
// ===== library: MasterCopy "S7-1500_LAnyAxis_Blocks (Drop in folder "Program blocks")" =====

// folder: LAnyAxis_Blocks

FUNCTION_BLOCK "LAnyAxis_MC_Power"   // FB30000, SCL
TITLE = LAnyAxis_MC_Power
{ S7_Optimized_Access := 'TRUE' }
AUTHOR : tech.team.motioncontrol@siemens.com
FAMILY : AnyAxis
VERSION : 1.0
// Support: tech.team.motioncontrol@siemens.com 
// See corresponding MC_ instruction in TIA Portal help (information system)
   VAR_INPUT
      Axis : DB_ANY;   // See corresponding parameter of MC_ instruction in TIA Portal help (information system)
      Enable : Bool;   // See corresponding parameter of MC_ instruction in TIA Portal help (information system)
      StartMode : DInt := 1;   // See corresponding parameter of MC_ instruction in TIA Portal help (information system)
      StopMode : Int;   // See corresponding parameter of MC_ instruction in TIA Portal help (information system)
   END_VAR
   VAR_OUTPUT
      Status : Bool;   // See corresponding parameter of MC_ instruction in TIA Portal help (information system)
      Busy : Bool;   // See corresponding parameter of MC_ instruction in TIA Portal help (information system)
      Error : Bool;   // See corresponding parameter of MC_ instruction in TIA Portal help (information system)
      ErrorID : Word;   // See corresponding parameter of MC_ instruction in TIA Portal help (information system)
   END_VAR
   VAR
      instMC : MC_POWER;   // Instance of MC_Instruction
      statAxis : DB_ANY;   // Internal variable of axis
      statAxisType : Int;   // Actual state / axis type
   END_VAR
   VAR CONSTANT
      ERROR_INVALID_TECHNOLOGY_OBJECT : Word := 16#8002;   // See corresponding parameter of MC_ instruction in TIA Portal help (information system)
      IDLE : Int := 0;   // State idle
      INVALID_AXIS : Int := -1;   // Axis type: Invalid
      EXTERNAL_ENCODER : Int := 1;   // Axis type: External encoder
      SPEED_AXIS : Int := 2;   // Axis type: Speed axis
      POSITIONING_AXIS : Int := 3;   // Axis type: Positioning axis
      SYNCHRONOUS_AXIS : Int := 4;   // Axis type: Synchronous axis
   END_VAR
BEGIN
   REGION HEADER
     //================================================================================
     // SIEMENS AG
     // (c)Copyright 2020 All Rights Reserved
     //--------------------------------------------------------------------------------
     // Library: LAnyAxis 
     // Tested with: S7-1515-2 PN
     // Engineering: TIA Portal V16
     // Restrictions: -
     // Requirements: S7-1500 FW 2.8.1
     // Functionality: Conversion DB_ANY --> TO_Axis
     // Support: tech.team.motioncontrol@siemens.com
     // Note: Parameter comments are only available in language 'English (United States)'
     //--------------------------------------------------------------------------------
     // Change log table:
     // Version  Date        Expert in charge  Changes applied
     // 01.00.00 10.03.2020  RS                First released version
     //================================================================================
   END_REGION

   REGION ENABLE
     IF (#statAxisType = #IDLE) AND #Enable THEN
       // Check axis type
       CASE TypeOfDB(#Axis) OF
         TO_POSITIONINGAXIS:
           #statAxisType := #POSITIONING_AXIS;
           #statAxis := #Axis;

         TO_SYNCHRONOUSAXIS:
           #statAxisType := #SYNCHRONOUS_AXIS;
           #statAxis := #Axis;

         TO_SPEEDAXIS:
           #statAxisType := #SPEED_AXIS;
           #statAxis := #Axis;

         TO_EXTERNALENCODER:
           #statAxisType := #EXTERNAL_ENCODER;
           #statAxis := #Axis;
         ELSE
           #statAxisType := #INVALID_AXIS;
           #statAxis := 0;
       END_CASE;

     ELSIF NOT #Enable AND (#statAxisType = #INVALID_AXIS) THEN
       #statAxisType := #IDLE;

       // Outputs
       #Status := FALSE;
       #Busy := FALSE;
       #Error := FALSE;
       #ErrorID := 16#0000;
     END_IF;
   END_REGION

   CASE #statAxisType OF
     #IDLE:
       ;

     #POSITIONING_AXIS,
     #SYNCHRONOUS_AXIS,
     #SPEED_AXIS,
     #EXTERNAL_ENCODER:
       REGION VALID_AXIS
         // Inputs
         #instMC.Enable := #Enable;
         #instMC.StartMode := #StartMode;
         #instMC.StopMode := #StopMode;

         // Call of MC instruction
         CASE #statAxisType OF
           #POSITIONING_AXIS:
             "LAnyAxis_UnpubPowerPosAxis"(axis := #statAxis,
                                          instMC := #instMC);
           #SYNCHRONOUS_AXIS:
             "LAnyAxis_UnpubPowerSyncAxis"(axis := #statAxis,
                                           instMC := #instMC);
           #SPEED_AXIS:
             "LAnyAxis_UnpubPowerSpeedAxis"(axis := #statAxis,
                                            instMC := #instMC);
           #EXTERNAL_ENCODER:
             "LAnyAxis_UnpubPowerExtEncoder"(axis := #statAxis,
                                             instMC := #instMC);
         END_CASE;

         // Outputs
         #Status := #instMC.Status;
         #Busy := #instMC.Busy;
         #Error := #instMC.Error;
         #ErrorID := #instMC.ErrorId;

         // Status of MC instruction
         IF NOT #instMC.Busy
           AND NOT #instMC.Error
           AND NOT #instMC.Status
         THEN
           // Not active
           #statAxisType := #IDLE;
         END_IF;
       END_REGION

     ELSE
       REGION INVALID_AXIS
         // Outputs
         #Status := FALSE;
         #Busy := FALSE;
         #Error := TRUE;
         #ErrorID := #ERROR_INVALID_TECHNOLOGY_OBJECT;
       END_REGION
   END_CASE;
END_FUNCTION_BLOCK

FUNCTION_BLOCK "LAnyAxis_MC_Reset"   // FB30001, SCL
TITLE = LAnyAxis_MC_Reset
{ S7_Optimized_Access := 'TRUE' }
AUTHOR : tech.team.motioncontrol@siemens.com
FAMILY : AnyAxis
VERSION : 1.0
// Support: tech.team.motioncontrol@siemens.com 
// See corresponding MC_ instruction in TIA Portal help (information system)
   VAR_INPUT
      Axis : DB_ANY;   // See corresponding parameter of MC_ instruction in TIA Portal help (information system)
      Execute : Bool;   // See corresponding parameter of MC_ instruction in TIA Portal help (information system)
      Restart : Bool;   // See corresponding parameter of MC_ instruction in TIA Portal help (information system)
   END_VAR
   VAR_OUTPUT
      Done : Bool;   // See corresponding parameter of MC_ instruction in TIA Portal help (information system)
      Busy : Bool;   // See corresponding parameter of MC_ instruction in TIA Portal help (information system)
      CommandAborted : Bool;   // See corresponding parameter of MC_ instruction in TIA Portal help (information system)
      Error : Bool;   // See corresponding parameter of MC_ instruction in TIA Portal help (information system)
      ErrorID : Word;   // See corresponding parameter of MC_ instruction in TIA Portal help (information system)
   END_VAR
   VAR
      instMC : MC_RESET;   // Instance of MC_Instruction
      statExecuteOld : Bool;   // Old value of execute
      statAxis : DB_ANY;   // Internal variable of axis
      statAxisType : Int;   // Actual state / axis type
   END_VAR
   VAR CONSTANT
      ERROR_INVALID_TECHNOLOGY_OBJECT : Word := 16#8002;   // See corresponding parameter of MC_ instruction in TIA Portal help (information system)
      IDLE : Int := 0;   // State idle
      INVALID_AXIS : Int := -1;   // Axis type: Invalid
      EXTERNAL_ENCODER : Int := 1;   // Axis type: External encoder
      SPEED_AXIS : Int := 2;   // Axis type: Speed axis
      POSITIONING_AXIS : Int := 3;   // Axis type: Positioning axis
      SYNCHRONOUS_AXIS : Int := 4;   // Axis type: Synchronous axis
      PROXY : Int := 5;   // Axis type: Leading axis proxy
   END_VAR
BEGIN
   REGION HEADER
     //================================================================================
     // SIEMENS AG
     // (c)Copyright 2020 All Rights Reserved
     //--------------------------------------------------------------------------------
     // Library: LAnyAxis 
     // Tested with: S7-1515-2 PN
     // Engineering: TIA Portal V16
     // Restrictions: -
     // Requirements: S7-1500 FW 2.8.1
     // Functionality: Conversion DB_ANY --> TO_Axis
     // Support: tech.team.motioncontrol@siemens.com
     // Note: Parameter comments are only available in language 'English (United States)'
     //--------------------------------------------------------------------------------
     // Change log table:
     // Version  Date        Expert in charge  Changes applied
     // 01.00.00 10.03.2020  RS                First released version
     //================================================================================
   END_REGION

   REGION EXECUTE
     IF #Execute AND NOT #statExecuteOld THEN
       // Copy parameter
       #instMC.Restart := #Restart;

       // Check axis type
       CASE TypeOfDB(#Axis) OF
         TO_POSITIONINGAXIS:
           #statAxisType := #POSITIONING_AXIS;
           #statAxis := #Axis;

         TO_SYNCHRONOUSAXIS:
           #statAxisType := #SYNCHRONOUS_AXIS;
           #statAxis := #Axis;

         TO_EXTERNALENCODER:
           #statAxisType := #EXTERNAL_ENCODER;
           #statAxis := #Axis;

         TO_SPEEDAXIS:
           #statAxisType := #SPEED_AXIS;
           #statAxis := #Axis;

         ELSE
           #statAxisType := #INVALID_AXIS;
           #statAxis := 0;
       END_CASE;

     ELSIF NOT #Execute AND (#statAxisType = #INVALID_AXIS) THEN
       #statAxisType := #IDLE;

       // Outputs
       #Done := FALSE;
       #Busy := FALSE;
       #CommandAborted := FALSE;
       #Error := FALSE;
       #ErrorID := 16#0000;
     END_IF;

     // Edge detection
     #statExecuteOld := #Execute;
   END_REGION

   CASE #statAxisType OF
     #IDLE:
       ;

     #POSITIONING_AXIS,
     #SYNCHRONOUS_AXIS,
     #SPEED_AXIS,
     #EXTERNAL_ENCODER,
     #PROXY:
       REGION VALID_AXIS
         // Inputs
         #instMC.Execute := #Execute;

         // Call of MC instruction
         CASE #statAxisType OF
           #POSITIONING_AXIS:
             "LAnyAxis_UnpubResetPosAxis"(axis := #statAxis,
                                          instMC := #instMC);
           #SYNCHRONOUS_AXIS:
             "LAnyAxis_UnpubResetSyncAxis"(axis := #statAxis,
                                           instMC := #instMC);
           #SPEED_AXIS:
             "LAnyAxis_UnpubResetSpeedAxis"(axis := #statAxis,
                                            instMC := #instMC);
           #EXTERNAL_ENCODER:
             "LAnyAxis_UnpubResetExtEncoder"(axis := #statAxis,
                                             instMC := #instMC);
         END_CASE;

         // Outputs
         #Done := #instMC.Done;
         #Busy := #instMC.Busy;
         #CommandAborted := #instMC.CommandAborted;
         #Error := #instMC.Error;
         #ErrorID := #instMC.ErrorId;

         // Status of MC instruction
         IF NOT #instMC.Done
           AND NOT #instMC.Busy
           AND NOT #instMC.CommandAborted
           AND NOT #instMC.Error
         THEN
           // Not active
           #statAxisType := #IDLE;
         END_IF;
       END_REGION

     ELSE
       REGION INVALID_AXIS
         // Outputs
         #Done := FALSE;
         #Busy := FALSE;
         #CommandAborted := FALSE;
         #Error := TRUE;
         #ErrorID := #ERROR_INVALID_TECHNOLOGY_OBJECT;
       END_REGION
   END_CASE;
END_FUNCTION_BLOCK

FUNCTION_BLOCK "LAnyAxis_MC_Home"   // FB30002, SCL
TITLE = LAnyAxis_MC_Home
{ S7_Optimized_Access := 'TRUE' }
AUTHOR : tech.team.motioncontrol@siemens.com
FAMILY : AnyAxis
VERSION : 1.0
// Support: tech.team.motioncontrol@siemens.com 
// See corresponding MC_ instruction in TIA Portal help (information system)
   VAR_INPUT
      Axis : DB_ANY;   // See corresponding parameter of MC_ instruction in TIA Portal help (information system)
      Execute : Bool;   // See corresponding parameter of MC_ instruction in TIA Portal help (information system)
      Position : LReal;   // See corresponding parameter of MC_ instruction in TIA Portal help (information system)
      Mode : Int;   // See corresponding parameter of MC_ instruction in TIA Portal help (information system)
   END_VAR
   VAR_OUTPUT
      ReferenceMarkPosition : LReal;   // See corresponding parameter of MC_ instruction in TIA Portal help (information system)
      Done : Bool;   // See corresponding parameter of MC_ instruction in TIA Portal help (information system)
      Busy : Bool;   // See corresponding parameter of MC_ instruction in TIA Portal help (information system)
      CommandAborted : Bool;   // See corresponding parameter of MC_ instruction in TIA Portal help (information system)
      Error : Bool;   // See corresponding parameter of MC_ instruction in TIA Portal help (information system)
      ErrorID : Word;   // See corresponding parameter of MC_ instruction in TIA Portal help (information system)
   END_VAR
   VAR
      instMC : MC_HOME;   // Instance of MC_Instruction
      statExecuteOld : Bool;   // Old value of execute
      statAxis : DB_ANY;   // Internal variable of axis
      statAxisType : Int;   // Actual state / axis type
   END_VAR
   VAR CONSTANT
      ERROR_INVALID_TECHNOLOGY_OBJECT : Word := 16#8002;   // See corresponding parameter of MC_ instruction in TIA Portal help (information system)
      IDLE : Int := 0;   // State idle
      INVALID_AXIS : Int := -1;   // Axis type: Invalid
      EXTERNAL_ENCODER : Int := 1;   // Axis type: External encoder
      POSITIONING_AXIS : Int := 3;   // Axis type: Positioning axis
      SYNCHRONOUS_AXIS : Int := 4;   // Axis type: Synchronous axis
   END_VAR
BEGIN
   REGION HEADER
     //================================================================================
     // SIEMENS AG
     // (c)Copyright 2020 All Rights Reserved
     //--------------------------------------------------------------------------------
     // Library: LAnyAxis 
     // Tested with: S7-1515-2 PN
     // Engineering: TIA Portal V16
     // Restrictions: -
     // Requirements: S7-1500 FW 2.8.1
     // Functionality: Conversion DB_ANY --> TO_Axis
     // Support: tech.team.motioncontrol@siemens.com
     // Note: Parameter comments are only available in language 'English (United States)'
     //--------------------------------------------------------------------------------
     // Change log table:
     // Version  Date        Expert in charge  Changes applied
     // 01.00.00 10.03.2020  RS                First released version
     //================================================================================
   END_REGION

   REGION EXECUTE
     IF #Execute AND NOT #statExecuteOld THEN
       // Copy parameter
       #instMC.Position := #Position;
       #instMC.Mode := #Mode;

       // Check axis type
       CASE TypeOfDB(#Axis) OF
         TO_POSITIONINGAXIS:
           #statAxisType := #POSITIONING_AXIS;
           #statAxis := #Axis;

         TO_SYNCHRONOUSAXIS:
           #statAxisType := #SYNCHRONOUS_AXIS;
           #statAxis := #Axis;

         TO_EXTERNALENCODER:
           #statAxisType := #EXTERNAL_ENCODER;
           #statAxis := #Axis;

         ELSE
           #statAxisType := #INVALID_AXIS;
           #statAxis := 0;
       END_CASE;

     ELSIF NOT #Execute AND (#statAxisType = #INVALID_AXIS) THEN
       #statAxisType := #IDLE;

       // Outputs
       #Done := FALSE;
       #Busy := FALSE;
       #CommandAborted := FALSE;
       #Error := FALSE;
       #ErrorID := 16#0000;
     END_IF;

     // Edge detection
     #statExecuteOld := #Execute;
   END_REGION

   CASE #statAxisType OF
     #IDLE:
       ;

     #POSITIONING_AXIS,
     #SYNCHRONOUS_AXIS,
     #EXTERNAL_ENCODER:
       REGION VALID_AXIS
         // Inputs
         #instMC.Execute := #Execute;

         // Call of MC instruction
         CASE #statAxisType OF
           #POSITIONING_AXIS:
             "LAnyAxis_UnpubHomePosAxis"(axis := #statAxis,
                                         instMC := #instMC);
           #SYNCHRONOUS_AXIS:
             "LAnyAxis_UnpubHomeSyncAxis"(axis := #statAxis,
                                          instMC := #instMC);
           #EXTERNAL_ENCODER:
             "LAnyAxis_UnpubHomeExtEncoder"(axis := #statAxis,
                                            instMC := #instMC);
         END_CASE;

         // Outputs
         #ReferenceMarkPosition := #instMC.ReferenceMarkPosition;
         #Done := #instMC.Done;
         #Busy := #instMC.Busy;
         #CommandAborted := #instMC.CommandAborted;
         #Error := #instMC.Error;
         #ErrorID := #instMC.ErrorId;

         // Status of MC instruction
         IF NOT #instMC.Done
           AND NOT #instMC.Busy
           AND NOT #instMC.CommandAborted
           AND NOT #instMC.Error
         THEN
           // Not active
           #statAxisType := #IDLE;
         END_IF;
       END_REGION

     ELSE
       REGION INVALID_AXIS
         // Outputs
         #Done := FALSE;
         #Busy := FALSE;
         #CommandAborted := FALSE;
         #Error := TRUE;
         #ErrorID := #ERROR_INVALID_TECHNOLOGY_OBJECT;
       END_REGION
   END_CASE;
END_FUNCTION_BLOCK

FUNCTION_BLOCK "LAnyAxis_MC_Halt"   // FB30003, SCL
TITLE = LAnyAxis_MC_Halt
{ S7_Optimized_Access := 'TRUE' }
AUTHOR : tech.team.motioncontrol@siemens.com
FAMILY : AnyAxis
VERSION : 1.0
// Support: tech.team.motioncontrol@siemens.com 
// See corresponding MC_ instruction in TIA Portal help (information system)
   VAR_INPUT
      Axis : DB_ANY;   // See corresponding parameter of MC_ instruction in TIA Portal help (information system)
      Execute : Bool;   // See corresponding parameter of MC_ instruction in TIA Portal help (information system)
      Deceleration : LReal := -1.0;   // See corresponding parameter of MC_ instruction in TIA Portal help (information system)
      Jerk : LReal := -1.0;   // See corresponding parameter of MC_ instruction in TIA Portal help (information system)
      AbortAcceleration : Bool;   // See corresponding parameter of MC_ instruction in TIA Portal help (information system)
   END_VAR
   VAR_OUTPUT
      Done : Bool;   // See corresponding parameter of MC_ instruction in TIA Portal help (information system)
      Busy : Bool;   // See corresponding parameter of MC_ instruction in TIA Portal help (information system)
      CommandAborted : Bool;   // See corresponding parameter of MC_ instruction in TIA Portal help (information system)
      Error : Bool;   // See corresponding parameter of MC_ instruction in TIA Portal help (information system)
      ErrorID : Word;   // See corresponding parameter of MC_ instruction in TIA Portal help (information system)
   END_VAR
   VAR
      instMC : MC_HALT;   // Instance of MC_Instruction
      statExecuteOld : Bool;   // Old value of execute
      statAxis : DB_ANY;   // Internal variable of axis
      statAxisType : Int;   // Actual state / axis type
   END_VAR
   VAR CONSTANT
      ERROR_INVALID_TECHNOLOGY_OBJECT : Word := 16#8002;   // See corresponding parameter of MC_ instruction in TIA Portal help (information system)
      IDLE : Int := 0;   // State idle
      INVALID_AXIS : Int := -1;   // Axis type: Invalid
      SPEED_AXIS : Int := 2;   // Axis type: Speed axis
      POSITIONING_AXIS : Int := 3;   // Axis type: Positioning axis
      SYNCHRONOUS_AXIS : Int := 4;   // Axis type: Synchronous axis
   END_VAR
BEGIN
   REGION HEADER
     //================================================================================
     // SIEMENS AG
     // (c)Copyright 2020 All Rights Reserved
     //--------------------------------------------------------------------------------
     // Library: LAnyAxis 
     // Tested with: S7-1515-2 PN
     // Engineering: TIA Portal V16
     // Restrictions: -
     // Requirements: S7-1500 FW 2.8.1
     // Functionality: Conversion DB_ANY --> TO_Axis
     // Support: tech.team.motioncontrol@siemens.com
     // Note: Parameter comments are only available in language 'English (United States)'
     //--------------------------------------------------------------------------------
     // Change log table:
     // Version  Date        Expert in charge  Changes applied
     // 01.00.00 10.03.2020  RS                First released version
     //================================================================================
   END_REGION

   REGION EXECUTE
     IF #Execute AND NOT #statExecuteOld THEN
       // Copy parameter
       #instMC.Deceleration := #Deceleration;
       #instMC.Jerk := #Jerk;
       #instMC.AbortAcceleration := #AbortAcceleration;

       // Check axis type
       CASE TypeOfDB(#Axis) OF
         TO_POSITIONINGAXIS:
           #statAxisType := #POSITIONING_AXIS;
           #statAxis := #Axis;

         TO_SYNCHRONOUSAXIS:
           #statAxisType := #SYNCHRONOUS_AXIS;
           #statAxis := #Axis;

         TO_SPEEDAXIS:
           #statAxisType := #SPEED_AXIS;
           #statAxis := #Axis;

         ELSE
           #statAxisType := #INVALID_AXIS;
           #statAxis := 0;
       END_CASE;

     ELSIF NOT #Execute AND (#statAxisType = #INVALID_AXIS) THEN
       #statAxisType := #IDLE;

       // Outputs
       #Done := FALSE;
       #Busy := FALSE;
       #CommandAborted := FALSE;
       #Error := FALSE;
       #ErrorID := 16#0000;
     END_IF;

     // Edge detection
     #statExecuteOld := #Execute;
   END_REGION

   CASE #statAxisType OF
     #IDLE:
       ;

     #POSITIONING_AXIS,
     #SYNCHRONOUS_AXIS,
     #SPEED_AXIS:
       REGION VALID_AXIS
         // Inputs
         #instMC.Execute := #Execute;

         // Call of MC instruction
         CASE #statAxisType OF
           #POSITIONING_AXIS:
             "LAnyAxis_UnpubHaltPosAxis"(axis := #statAxis,
                                         instMC := #instMC);
           #SYNCHRONOUS_AXIS:
             "LAnyAxis_UnpubHaltSyncAxis"(axis := #statAxis,
                                          instMC := #instMC);
           #SPEED_AXIS:
             #instMC(Axis := #statAxis);
         END_CASE;

         // Outputs
         #Done := #instMC.Done;
         #Busy := #instMC.Busy;
         #CommandAborted := #instMC.CommandAborted;
         #Error := #instMC.Error;
         #ErrorID := #instMC.ErrorId;

         // Status of MC instruction
         IF NOT #instMC.Done
           AND NOT #instMC.Busy
           AND NOT #instMC.CommandAborted
           AND NOT #instMC.Error
         THEN
           // Not active
           #statAxisType := #IDLE;
         END_IF;
       END_REGION

     ELSE
       REGION INVALID_AXIS
         // Outputs
         #Done := FALSE;
         #Busy := FALSE;
         #CommandAborted := FALSE;
         #Error := TRUE;
         #ErrorID := #ERROR_INVALID_TECHNOLOGY_OBJECT;
       END_REGION
   END_CASE;
END_FUNCTION_BLOCK

FUNCTION_BLOCK "LAnyAxis_MC_MoveAbsolute"   // FB30004, SCL
TITLE = LAnyAxis_MC_MoveAbsolute
{ S7_Optimized_Access := 'TRUE' }
AUTHOR : tech.team.motioncontrol@siemens.com
FAMILY : AnyAxis
VERSION : 1.0
// Support: tech.team.motioncontrol@siemens.com 
// See corresponding MC_ instruction in TIA Portal help (information system)
   VAR_INPUT
      Axis : DB_ANY;   // See corresponding parameter of MC_ instruction in TIA Portal help (information system)
      Execute : Bool;   // See corresponding parameter of MC_ instruction in TIA Portal help (information system)
      Position : LReal;   // See corresponding parameter of MC_ instruction in TIA Portal help (information system)
      Velocity : LReal := -1.0;   // See corresponding parameter of MC_ instruction in TIA Portal help (information system)
      Acceleration : LReal := -1.0;   // See corresponding parameter of MC_ instruction in TIA Portal help (information system)
      Deceleration : LReal := -1.0;   // See corresponding parameter of MC_ instruction in TIA Portal help (information system)
      Jerk : LReal := -1.0;   // See corresponding parameter of MC_ instruction in TIA Portal help (information system)
      Direction : Int := 1;   // See corresponding parameter of MC_ instruction in TIA Portal help (information system)
   END_VAR
   VAR_OUTPUT
      Done : Bool;   // See corresponding parameter of MC_ instruction in TIA Portal help (information system)
      Busy : Bool;   // See corresponding parameter of MC_ instruction in TIA Portal help (information system)
      CommandAborted : Bool;   // See corresponding parameter of MC_ instruction in TIA Portal help (information system)
      Error : Bool;   // See corresponding parameter of MC_ instruction in TIA Portal help (information system)
      ErrorID : Word;   // See corresponding parameter of MC_ instruction in TIA Portal help (information system)
   END_VAR
   VAR
      instMC : MC_MOVEABSOLUTE;   // Instance of MC_Instruction
      statExecuteOld : Bool;   // Old value of execute
      statAxis : DB_ANY;   // Internal variable of axis
      statAxisType : Int;   // Actual state / axis type
   END_VAR
   VAR CONSTANT
      ERROR_INVALID_TECHNOLOGY_OBJECT : Word := 16#8002;   // See corresponding parameter of MC_ instruction in TIA Portal help (information system)
      IDLE : Int := 0;   // State idle
      INVALID_AXIS : Int := -1;   // Axis type: Invalid
      EXTERNAL_ENCODER : Int := 1;   // Axis type: External encoder
      POSITIONING_AXIS : Int := 3;   // Axis type: Positioning axis
      SYNCHRONOUS_AXIS : Int := 4;   // Axis type: Synchronous axis
   END_VAR
BEGIN
   REGION HEADER
     //================================================================================
     // SIEMENS AG
     // (c)Copyright 2020 All Rights Reserved
     //--------------------------------------------------------------------------------
     // Library: LAnyAxis 
     // Tested with: S7-1515-2 PN
     // Engineering: TIA Portal V16
     // Restrictions: -
     // Requirements: S7-1500 FW 2.8.1
     // Functionality: Conversion DB_ANY --> TO_Axis
     // Support: tech.team.motioncontrol@siemens.com
     // Note: Parameter comments are only available in language 'English (United States)'
     //--------------------------------------------------------------------------------
     // Change log table:
     // Version  Date        Expert in charge  Changes applied
     // 01.00.00 10.03.2020  RS                First released version
     //================================================================================
   END_REGION

   REGION EXECUTE
     IF #Execute AND NOT #statExecuteOld THEN
       // Copy parameter
       #instMC.Position := #Position;
       #instMC.Velocity := #Velocity;
       #instMC.Acceleration := #Acceleration;
       #instMC.Deceleration := #Deceleration;
       #instMC.Jerk := #Jerk;
       #instMC.Direction := #Direction;

       // Check axis type
       CASE TypeOfDB(#Axis) OF
         TO_POSITIONINGAXIS:
           #statAxisType := #POSITIONING_AXIS;
           #statAxis := #Axis;

         TO_SYNCHRONOUSAXIS:
           #statAxisType := #SYNCHRONOUS_AXIS;
           #statAxis := #Axis;

         ELSE
           #statAxisType := #INVALID_AXIS;
           #statAxis := 0;
       END_CASE;

     ELSIF NOT #Execute AND (#statAxisType = #INVALID_AXIS) THEN
       #statAxisType := #IDLE;

       // Outputs
       #Done := FALSE;
       #Busy := FALSE;
       #CommandAborted := FALSE;
       #Error := FALSE;
       #ErrorID := 16#0000;
     END_IF;

     // Edge detection
     #statExecuteOld := #Execute;
   END_REGION

   CASE #statAxisType OF
     #IDLE:
       ;

     #POSITIONING_AXIS,
     #SYNCHRONOUS_AXIS:
       REGION VALID_AXIS
         // Inputs
         #instMC.Execute := #Execute;

         // Call of MC instruction
         CASE #statAxisType OF
           #POSITIONING_AXIS:
             #instMC(Axis := #statAxis);
           #SYNCHRONOUS_AXIS:
             "LAnyAxis_UnpubMoveAbsoluteSyncAxis"(axis := #statAxis,
                                                  instMC := #instMC);
         END_CASE;

         // Outputs
         #Done := #instMC.Done;
         #Busy := #instMC.Busy;
         #CommandAborted := #instMC.CommandAborted;
         #Error := #instMC.Error;
         #ErrorID := #instMC.ErrorId;

         // Status of MC instruction
         IF NOT #instMC.Done
           AND NOT #instMC.Busy
           AND NOT #instMC.CommandAborted
           AND NOT #instMC.Error
         THEN
           // Not active
           #statAxisType := #IDLE;
         END_IF;
       END_REGION

     ELSE
       REGION INVALID_AXIS
         // Outputs
         #Done := FALSE;
         #Busy := FALSE;
         #CommandAborted := FALSE;
         #Error := TRUE;
         #ErrorID := #ERROR_INVALID_TECHNOLOGY_OBJECT;
       END_REGION
   END_CASE;
END_FUNCTION_BLOCK

FUNCTION_BLOCK "LAnyAxis_MC_MoveRelative"   // FB30005, SCL
TITLE = LAnyAxis_MC_MoveRelative
{ S7_Optimized_Access := 'TRUE' }
AUTHOR : tech.team.motioncontrol@siemens.com
FAMILY : AnyAxis
VERSION : 1.0
// Support: tech.team.motioncontrol@siemens.com 
// See corresponding MC_ instruction in TIA Portal help (information system)
   VAR_INPUT
      Axis : DB_ANY;   // See corresponding parameter of MC_ instruction in TIA Portal help (information system)
      Execute : Bool;   // See corresponding parameter of MC_ instruction in TIA Portal help (information system)
      Distance : LReal;   // See corresponding parameter of MC_ instruction in TIA Portal help (information system)
      Velocity : LReal := -1.0;   // See corresponding parameter of MC_ instruction in TIA Portal help (information system)
      Acceleration : LReal := -1.0;   // See corresponding parameter of MC_ instruction in TIA Portal help (information system)
      Deceleration : LReal := -1.0;   // See corresponding parameter of MC_ instruction in TIA Portal help (information system)
      Jerk : LReal := -1.0;   // See corresponding parameter of MC_ instruction in TIA Portal help (information system)
   END_VAR
   VAR_OUTPUT
      Done : Bool;   // See corresponding parameter of MC_ instruction in TIA Portal help (information system)
      Busy : Bool;   // See corresponding parameter of MC_ instruction in TIA Portal help (information system)
      CommandAborted : Bool;   // See corresponding parameter of MC_ instruction in TIA Portal help (information system)
      Error : Bool;   // See corresponding parameter of MC_ instruction in TIA Portal help (information system)
      ErrorID : Word;   // See corresponding parameter of MC_ instruction in TIA Portal help (information system)
   END_VAR
   VAR
      instMC : MC_MOVERELATIVE;   // Instance of MC_Instruction
      statExecuteOld : Bool;   // Old value of execute
      statAxis : DB_ANY;   // Internal variable of axis
      statAxisType : Int;   // Actual state / axis type
   END_VAR
   VAR CONSTANT
      ERROR_INVALID_TECHNOLOGY_OBJECT : Word := 16#8002;   // See corresponding parameter of MC_ instruction in TIA Portal help (information system)
      IDLE : Int := 0;   // State idle
      INVALID_AXIS : Int := -1;   // Axis type: Invalid
      POSITIONING_AXIS : Int := 3;   // Axis type: Positioning axis
      SYNCHRONOUS_AXIS : Int := 4;   // Axis type: Synchronous axis
   END_VAR
BEGIN
   REGION HEADER
     //================================================================================
     // SIEMENS AG
     // (c)Copyright 2020 All Rights Reserved
     //--------------------------------------------------------------------------------
     // Library: LAnyAxis 
     // Tested with: S7-1515-2 PN
     // Engineering: TIA Portal V16
     // Restrictions: -
     // Requirements: S7-1500 FW 2.8.1
     // Functionality: Conversion DB_ANY --> TO_Axis
     // Support: tech.team.motioncontrol@siemens.com
     // Note: Parameter comments are only available in language 'English (United States)'
     //--------------------------------------------------------------------------------
     // Change log table:
     // Version  Date        Expert in charge  Changes applied
     // 01.00.00 10.03.2020  RS                First released version
     //================================================================================
   END_REGION

   REGION EXECUTE
     IF #Execute AND NOT #statExecuteOld THEN
       // Copy parameter
       #instMC.Distance := #Distance;
       #instMC.Velocity := #Velocity;
       #instMC.Acceleration := #Acceleration;
       #instMC.Deceleration := #Deceleration;
       #instMC.Jerk := #Jerk;

       // Check axis type
       CASE TypeOfDB(#Axis) OF
         TO_POSITIONINGAXIS:
           #statAxisType := #POSITIONING_AXIS;
           #statAxis := #Axis;

         TO_SYNCHRONOUSAXIS:
           #statAxisType := #SYNCHRONOUS_AXIS;
           #statAxis := #Axis;

         ELSE
           #statAxisType := #INVALID_AXIS;
           #statAxis := 0;
       END_CASE;

     ELSIF NOT #Execute AND (#statAxisType = #INVALID_AXIS) THEN
       #statAxisType := #IDLE;

       // Outputs
       #Done := FALSE;
       #Busy := FALSE;
       #CommandAborted := FALSE;
       #Error := FALSE;
       #ErrorID := 16#0000;
     END_IF;

     // Edge detection
     #statExecuteOld := #Execute;
   END_REGION

   CASE #statAxisType OF
     #IDLE:
       ;

     #POSITIONING_AXIS,
     #SYNCHRONOUS_AXIS:
       REGION VALID_AXIS
         // Inputs
         #instMC.Execute := #Execute;

         // Call of MC instruction
         CASE #statAxisType OF
           #POSITIONING_AXIS:
             #instMC(Axis := #statAxis);
           #SYNCHRONOUS_AXIS:
             "LAnyAxis_UnpubMoveRelativeSyncAxis"(axis := #statAxis,
                                                  instMC := #instMC);
         END_CASE;

         // Outputs
         #Done := #instMC.Done;
         #Busy := #instMC.Busy;
         #CommandAborted := #instMC.CommandAborted;
         #Error := #instMC.Error;
         #ErrorID := #instMC.ErrorId;

         // Status of MC instruction
         IF NOT #instMC.Done
           AND NOT #instMC.Busy
           AND NOT #instMC.CommandAborted
           AND NOT #instMC.Error
         THEN
           // Not active
           #statAxisType := #IDLE;
         END_IF;
       END_REGION

     ELSE
       REGION INVALID_AXIS
         // Outputs
         #Done := FALSE;
         #Busy := FALSE;
         #CommandAborted := FALSE;
         #Error := TRUE;
         #ErrorID := #ERROR_INVALID_TECHNOLOGY_OBJECT;
       END_REGION
   END_CASE;
END_FUNCTION_BLOCK

FUNCTION_BLOCK "LAnyAxis_MC_MoveVelocity"   // FB30006, SCL
TITLE = LAnyAxis_MC_MoveVelocity
{ S7_Optimized_Access := 'TRUE' }
AUTHOR : tech.team.motioncontrol@siemens.com
FAMILY : AnyAxis
VERSION : 1.0
// Support: tech.team.motioncontrol@siemens.com 
// See corresponding MC_ instruction in TIA Portal help (information system)
   VAR_INPUT
      Axis : DB_ANY;   // See corresponding parameter of MC_ instruction in TIA Portal help (information system)
      Execute : Bool;   // See corresponding parameter of MC_ instruction in TIA Portal help (information system)
      Velocity : LReal := 100.0;   // See corresponding parameter of MC_ instruction in TIA Portal help (information system)
      Acceleration : LReal := -1.0;   // See corresponding parameter of MC_ instruction in TIA Portal help (information system)
      Deceleration : LReal := -1.0;   // See corresponding parameter of MC_ instruction in TIA Portal help (information system)
      Jerk : LReal := -1.0;   // See corresponding parameter of MC_ instruction in TIA Portal help (information system)
      Direction : Int;   // See corresponding parameter of MC_ instruction in TIA Portal help (information system)
      Current : Bool;   // See corresponding parameter of MC_ instruction in TIA Portal help (information system)
      PositionControlled : Bool := TRUE;   // See corresponding parameter of MC_ instruction in TIA Portal help (information system)
   END_VAR
   VAR_OUTPUT
      InVelocity : Bool;   // See corresponding parameter of MC_ instruction in TIA Portal help (information system)
      Busy : Bool;   // See corresponding parameter of MC_ instruction in TIA Portal help (information system)
      CommandAborted : Bool;   // See corresponding parameter of MC_ instruction in TIA Portal help (information system)
      Error : Bool;   // See corresponding parameter of MC_ instruction in TIA Portal help (information system)
      ErrorID : Word;   // See corresponding parameter of MC_ instruction in TIA Portal help (information system)
   END_VAR
   VAR
      instMC : MC_MOVEVELOCITY;   // Instance of MC_Instruction
      statExecuteOld : Bool;   // Old value of execute
      statAxis : DB_ANY;   // Internal variable of axis
      statAxisType : Int;   // Actual state / axis type
   END_VAR
   VAR CONSTANT
      ERROR_INVALID_TECHNOLOGY_OBJECT : Word := 16#8002;   // See corresponding parameter of MC_ instruction in TIA Portal help (information system)
      IDLE : Int := 0;   // State idle
      INVALID_AXIS : Int := -1;   // Axis type: Invalid
      SPEED_AXIS : Int := 2;   // Axis type: Speed axis
      POSITIONING_AXIS : Int := 3;   // Axis type: Positioning axis
      SYNCHRONOUS_AXIS : Int := 4;   // Axis type: Synchronous axis
   END_VAR
BEGIN
   REGION HEADER
     //================================================================================
     // SIEMENS AG
     // (c)Copyright 2020 All Rights Reserved
     //--------------------------------------------------------------------------------
     // Library: LAnyAxis 
     // Tested with: S7-1515-2 PN
     // Engineering: TIA Portal V16
     // Restrictions: -
     // Requirements: S7-1500 FW 2.8.1
     // Functionality: Conversion DB_ANY --> TO_Axis
     // Support: tech.team.motioncontrol@siemens.com
     // Note: Parameter comments are only available in language 'English (United States)'
     //--------------------------------------------------------------------------------
     // Change log table:
     // Version  Date        Expert in charge  Changes applied
     // 01.00.00 10.03.2020  RS                First released version
     //================================================================================
   END_REGION

   REGION EXECUTE
     IF #Execute AND NOT #statExecuteOld THEN
       // Copy parameter
       #instMC.Velocity := #Velocity;
       #instMC.Acceleration := #Acceleration;
       #instMC.Deceleration := #Deceleration;
       #instMC.Jerk := #Jerk;
       #instMC.Direction := #Direction;
       #instMC.Current := #Current;
       #instMC.PositionControlled := #PositionControlled;

       // Check axis type
       CASE TypeOfDB(#Axis) OF
         TO_POSITIONINGAXIS:
           #statAxisType := #POSITIONING_AXIS;
           #statAxis := #Axis;

         TO_SYNCHRONOUSAXIS:
           #statAxisType := #SYNCHRONOUS_AXIS;
           #statAxis := #Axis;

         TO_SPEEDAXIS:
           #statAxisType := #SPEED_AXIS;
           #statAxis := #Axis;

         ELSE
           #statAxisType := #INVALID_AXIS;
           #statAxis := 0;
       END_CASE;

     ELSIF NOT #Execute AND (#statAxisType = #INVALID_AXIS) THEN
       #statAxisType := #IDLE;

       // Outputs
       #InVelocity := FALSE;
       #Busy := FALSE;
       #CommandAborted := FALSE;
       #Error := FALSE;
       #ErrorID := 16#0000;
     END_IF;

     // Edge detection
     #statExecuteOld := #Execute;
   END_REGION

   CASE #statAxisType OF
     #IDLE:
       ;

     #POSITIONING_AXIS,
     #SYNCHRONOUS_AXIS,
     #SPEED_AXIS:
       REGION VALID_AXIS
         // Inputs
         #instMC.Execute := #Execute;

         // Call of MC instruction
         CASE #statAxisType OF
           #POSITIONING_AXIS:
             "LAnyAxis_UnpubMoveVelocityPosAxis"(axis := #statAxis,
                                                 instMC := #instMC);
           #SYNCHRONOUS_AXIS:
             "LAnyAxis_UnpubMoveVelocitySyncAxis"(axis := #statAxis,
                                                  instMC := #instMC);
           #SPEED_AXIS:
             #instMC(Axis := #statAxis);
         END_CASE;

         // Outputs
         #InVelocity := #instMC.InVelocity;
         #Busy := #instMC.Busy;
         #CommandAborted := #instMC.CommandAborted;
         #Error := #instMC.Error;
         #ErrorID := #instMC.ErrorId;

         // Status of MC instruction
         IF NOT #instMC.Busy
           AND NOT #instMC.CommandAborted
           AND NOT #instMC.Error
         THEN
           // Not active
           #statAxisType := #IDLE;
         END_IF;
       END_REGION

     ELSE
       REGION INVALID_AXIS
         // Outputs
         #InVelocity := FALSE;
         #Busy := FALSE;
         #CommandAborted := FALSE;
         #Error := TRUE;
         #ErrorID := #ERROR_INVALID_TECHNOLOGY_OBJECT;
       END_REGION
   END_CASE;
END_FUNCTION_BLOCK

FUNCTION_BLOCK "LAnyAxis_MC_MoveJog"   // FB30007, SCL
TITLE = LAnyAxis_MC_MoveJog
{ S7_Optimized_Access := 'TRUE' }
AUTHOR : tech.team.motioncontrol@siemens.com
FAMILY : AnyAxis
VERSION : 1.0
// Support: tech.team.motioncontrol@siemens.com 
// See corresponding MC_ instruction in TIA Portal help (information system)
   VAR_INPUT
      Axis : DB_ANY;   // See corresponding parameter of MC_ instruction in TIA Portal help (information system)
      JogForward : Bool;   // See corresponding parameter of MC_ instruction in TIA Portal help (information system)
      JogBackward : Bool;   // See corresponding parameter of MC_ instruction in TIA Portal help (information system)
      Velocity : LReal := 100.0;   // See corresponding parameter of MC_ instruction in TIA Portal help (information system)
      Acceleration : LReal := -1.0;   // See corresponding parameter of MC_ instruction in TIA Portal help (information system)
      Deceleration : LReal := -1.0;   // See corresponding parameter of MC_ instruction in TIA Portal help (information system)
      Jerk : LReal := -1.0;   // See corresponding parameter of MC_ instruction in TIA Portal help (information system)
      PositionControlled : Bool := TRUE;   // See corresponding parameter of MC_ instruction in TIA Portal help (information system)
   END_VAR
   VAR_OUTPUT
      InVelocity : Bool;   // See corresponding parameter of MC_ instruction in TIA Portal help (information system)
      Busy : Bool;   // See corresponding parameter of MC_ instruction in TIA Portal help (information system)
      CommandAborted : Bool;   // See corresponding parameter of MC_ instruction in TIA Portal help (information system)
      Error : Bool;   // See corresponding parameter of MC_ instruction in TIA Portal help (information system)
      ErrorID : Word;   // See corresponding parameter of MC_ instruction in TIA Portal help (information system)
   END_VAR
   VAR
      instMC : MC_MOVEJOG;   // Instance of MC_Instruction
      statAxis : DB_ANY;   // Internal variable of axis
      statAxisType : Int;   // Actual state / axis type
   END_VAR
   VAR CONSTANT
      ERROR_INVALID_TECHNOLOGY_OBJECT : Word := 16#8002;   // See corresponding parameter of MC_ instruction in TIA Portal help (information system)
      IDLE : Int := 0;   // State idle
      INVALID_AXIS : Int := -1;   // Axis type: Invalid
      SPEED_AXIS : Int := 2;   // Axis type: Speed axis
      POSITIONING_AXIS : Int := 3;   // Axis type: Positioning axis
      SYNCHRONOUS_AXIS : Int := 4;   // Axis type: Synchronous axis
   END_VAR
BEGIN
   REGION HEADER
     //================================================================================
     // SIEMENS AG
     // (c)Copyright 2020 All Rights Reserved
     //--------------------------------------------------------------------------------
     // Library: LAnyAxis 
     // Tested with: S7-1515-2 PN
     // Engineering: TIA Portal V16
     // Restrictions: -
     // Requirements: S7-1500 FW 2.8.1
     // Functionality: Conversion DB_ANY --> TO_Axis
     // Support: tech.team.motioncontrol@siemens.com
     // Note: Parameter comments are only available in language 'English (United States)'
     //--------------------------------------------------------------------------------
     // Change log table:
     // Version  Date        Expert in charge  Changes applied
     // 01.00.00 10.03.2020  RS                First released version
     //================================================================================
   END_REGION

   REGION ENABLE
     IF (#statAxisType = #IDLE) AND (#JogForward OR #JogBackward) THEN
       // Check axis type
       CASE TypeOfDB(#Axis) OF
         TO_POSITIONINGAXIS:
           #statAxisType := #POSITIONING_AXIS;
           #statAxis := #Axis;

         TO_SYNCHRONOUSAXIS:
           #statAxisType := #SYNCHRONOUS_AXIS;
           #statAxis := #Axis;

         TO_SPEEDAXIS:
           #statAxisType := #SPEED_AXIS;
           #statAxis := #Axis;

         ELSE
           #statAxisType := #INVALID_AXIS;
           #statAxis := 0;
       END_CASE;

     ELSIF NOT #JogForward AND NOT #JogBackward AND (#statAxisType = #INVALID_AXIS) THEN
       #statAxisType := #IDLE;

       // Outputs
       #InVelocity := FALSE;
       #Busy := FALSE;
       #CommandAborted := FALSE;
       #Error := FALSE;
       #ErrorID := 16#0000;
     END_IF;
   END_REGION

   CASE #statAxisType OF
     #IDLE:
       ;

     #POSITIONING_AXIS,
     #SYNCHRONOUS_AXIS,
     #SPEED_AXIS:
       REGION VALID_AXIS
         // Inputs
         #instMC.JogForward := #JogForward;
         #instMC.JogBackward := #JogBackward;
         #instMC.Velocity := #Velocity;
         #instMC.Acceleration := #Acceleration;
         #instMC.Deceleration := #Deceleration;
         #instMC.Jerk := #Jerk;
         #instMC.PositionControlled := #PositionControlled;

         // Call of MC instruction
         CASE #statAxisType OF
           #POSITIONING_AXIS:
             "LAnyAxis_UnpubMoveJogPosAxis"(axis := #statAxis,
                                            instMC := #instMC);
           #SYNCHRONOUS_AXIS:
             "LAnyAxis_UnpubMoveJogSyncAxis"(axis := #statAxis,
                                             instMC := #instMC);
           #SPEED_AXIS:
             #instMC(Axis := #statAxis);
         END_CASE;

         // Outputs
         #InVelocity := #instMC.InVelocity;
         #Busy := #instMC.Busy;
         #CommandAborted := #instMC.CommandAborted;
         #Error := #instMC.Error;
         #ErrorID := #instMC.ErrorId;

         // Status of MC instruction
         IF NOT #instMC.Busy
           AND NOT #instMC.Error
           AND NOT #instMC.CommandAborted
         THEN
           // Not active
           #statAxisType := #IDLE;
         END_IF;
       END_REGION

     ELSE
       REGION INVALID_AXIS
         // Outputs
         #InVelocity := FALSE;
         #Busy := FALSE;
         #CommandAborted := FALSE;
         #Error := TRUE;
         #ErrorID := #ERROR_INVALID_TECHNOLOGY_OBJECT;
       END_REGION
   END_CASE;
END_FUNCTION_BLOCK

FUNCTION_BLOCK "LAnyAxis_MC_MoveSuperimposed"   // FB30008, SCL
TITLE = LAnyAxis_MC_MoveSuperimposed
{ S7_Optimized_Access := 'TRUE' }
AUTHOR : tech.team.motioncontrol@siemens.com
FAMILY : AnyAxis
VERSION : 1.0
// Support: tech.team.motioncontrol@siemens.com 
// See corresponding MC_ instruction in TIA Portal help (information system)
   VAR_INPUT
      Axis : DB_ANY;   // See corresponding parameter of MC_ instruction in TIA Portal help (information system)
      Execute : Bool;   // See corresponding parameter of MC_ instruction in TIA Portal help (information system)
      Distance : LReal;   // See corresponding parameter of MC_ instruction in TIA Portal help (information system)
      VelocityDiff : LReal := -1.0;   // See corresponding parameter of MC_ instruction in TIA Portal help (information system)
      Acceleration : LReal := -1.0;   // See corresponding parameter of MC_ instruction in TIA Portal help (information system)
      Deceleration : LReal := -1.0;   // See corresponding parameter of MC_ instruction in TIA Portal help (information system)
      Jerk : LReal := -1.0;   // See corresponding parameter of MC_ instruction in TIA Portal help (information system)
   END_VAR
   VAR_OUTPUT
      Done : Bool;   // See corresponding parameter of MC_ instruction in TIA Portal help (information system)
      Busy : Bool;   // See corresponding parameter of MC_ instruction in TIA Portal help (information system)
      CommandAborted : Bool;   // See corresponding parameter of MC_ instruction in TIA Portal help (information system)
      Error : Bool;   // See corresponding parameter of MC_ instruction in TIA Portal help (information system)
      ErrorID : Word;   // See corresponding parameter of MC_ instruction in TIA Portal help (information system)
   END_VAR
   VAR
      instMC : MC_MOVESUPERIMPOSED;   // Instance of MC_Instruction
      statExecuteOld : Bool;   // Old value of execute
      statAxis : DB_ANY;   // Internal variable of axis
      statAxisType : Int;   // Actual state / axis type
   END_VAR
   VAR CONSTANT
      ERROR_INVALID_TECHNOLOGY_OBJECT : Word := 16#8002;   // See corresponding parameter of MC_ instruction in TIA Portal help (information system)
      IDLE : Int := 0;   // State idle
      INVALID_AXIS : Int := -1;   // Axis type: Invalid
      POSITIONING_AXIS : Int := 3;   // Axis type: Positioning axis
      SYNCHRONOUS_AXIS : Int := 4;   // Axis type: Synchronous axis
   END_VAR
BEGIN
   REGION HEADER
     //================================================================================
     // SIEMENS AG
     // (c)Copyright 2020 All Rights Reserved
     //--------------------------------------------------------------------------------
     // Library: LAnyAxis 
     // Tested with: S7-1515-2 PN
     // Engineering: TIA Portal V16
     // Restrictions: -
     // Requirements: S7-1500 FW 2.8.1
     // Functionality: Conversion DB_ANY --> TO_Axis
     // Support: tech.team.motioncontrol@siemens.com
     // Note: Parameter comments are only available in language 'English (United States)'
     //--------------------------------------------------------------------------------
     // Change log table:
     // Version  Date        Expert in charge  Changes applied
     // 01.00.00 10.03.2020  RS                First released version
     //================================================================================
   END_REGION

   REGION EXECUTE
     IF #Execute AND NOT #statExecuteOld THEN
       // Copy parameter
       #instMC.Distance := #Distance;
       #instMC.VelocityDiff := #VelocityDiff;
       #instMC.Acceleration := #Acceleration;
       #instMC.Deceleration := #Deceleration;
       #instMC.Jerk := #Jerk;

       // Check axis type
       CASE TypeOfDB(#Axis) OF
         TO_POSITIONINGAXIS:
           #statAxisType := #POSITIONING_AXIS;
           #statAxis := #Axis;

         TO_SYNCHRONOUSAXIS:
           #statAxisType := #SYNCHRONOUS_AXIS;
           #statAxis := #Axis;

         ELSE
           #statAxisType := #INVALID_AXIS;
           #statAxis := 0;
       END_CASE;

     ELSIF NOT #Execute AND (#statAxisType = #INVALID_AXIS) THEN
       #statAxisType := #IDLE;

       // Outputs
       #Done := FALSE;
       #Busy := FALSE;
       #CommandAborted := FALSE;
       #Error := FALSE;
       #ErrorID := 16#0000;
     END_IF;

     // Edge detection
     #statExecuteOld := #Execute;
   END_REGION

   CASE #statAxisType OF
     #IDLE:
       ;

     #POSITIONING_AXIS,
     #SYNCHRONOUS_AXIS:
       REGION VALID_AXIS
         // Inputs
         #instMC.Execute := #Execute;

         // Call of MC instruction
         CASE #statAxisType OF
           #POSITIONING_AXIS:
             #instMC(Axis := #statAxis);
           #SYNCHRONOUS_AXIS:
             "LAnyAxis_UnpubMoveSuperimposedSyncAxis"(axis := #statAxis,
                                                      instMC := #instMC);
         END_CASE;

         // Outputs
         #Done := #instMC.Done;
         #Busy := #instMC.Busy;
         #CommandAborted := #instMC.CommandAborted;
         #Error := #instMC.Error;
         #ErrorID := #instMC.ErrorId;

         // Status of MC instruction
         IF NOT #instMC.Done
           AND NOT #instMC.Busy
           AND NOT #instMC.CommandAborted
           AND NOT #instMC.Error
         THEN
           // Not active
           #statAxisType := #IDLE;
         END_IF;
       END_REGION

     ELSE
       REGION INVALID_AXIS
         // Outputs
         #Done := FALSE;
         #Busy := FALSE;
         #CommandAborted := FALSE;
         #Error := TRUE;
         #ErrorID := #ERROR_INVALID_TECHNOLOGY_OBJECT;
       END_REGION
   END_CASE;
END_FUNCTION_BLOCK

FUNCTION_BLOCK "LAnyAxis_MC_SetAxisSTW"   // FB30011, SCL
TITLE = LAnyAxis_MC_SetAxisSTW
{ S7_Optimized_Access := 'TRUE' }
AUTHOR : tech.team.motioncontrol@siemens.com
FAMILY : AnyAxis
VERSION : 1.0
// Support: tech.team.motioncontrol@siemens.com 
// See corresponding MC_ instruction in TIA Portal help (information system)
   VAR_INPUT
      Axis : DB_ANY;   // See corresponding parameter of MC_ instruction in TIA Portal help (information system)
      Execute : Bool;   // See corresponding parameter of MC_ instruction in TIA Portal help (information system)
      STW1 : Word;   // See corresponding parameter of MC_ instruction in TIA Portal help (information system)
      STW1BitMask : Word;   // See corresponding parameter of MC_ instruction in TIA Portal help (information system)
      STW2 : Word;   // See corresponding parameter of MC_ instruction in TIA Portal help (information system)
      STW2BitMask : Word;   // See corresponding parameter of MC_ instruction in TIA Portal help (information system)
   END_VAR
   VAR_OUTPUT
      Done : Bool;   // See corresponding parameter of MC_ instruction in TIA Portal help (information system)
      Busy : Bool;   // See corresponding parameter of MC_ instruction in TIA Portal help (information system)
      CommandAborted : Bool;   // See corresponding parameter of MC_ instruction in TIA Portal help (information system)
      Error : Bool;   // See corresponding parameter of MC_ instruction in TIA Portal help (information system)
      ErrorID : Word;   // See corresponding parameter of MC_ instruction in TIA Portal help (information system)
   END_VAR
   VAR
      instMC : MC_SETAXISSTW;   // Instance of MC_Instruction
      statExecuteOld : Bool;   // Old value of execute
      statAxis : DB_ANY;   // Internal variable of axis
      statAxisType : Int;   // Actual state / axis type
   END_VAR
   VAR CONSTANT
      ERROR_INVALID_TECHNOLOGY_OBJECT : Word := 16#8002;   // See corresponding parameter of MC_ instruction in TIA Portal help (information system)
      IDLE : Int := 0;   // State idle
      INVALID_AXIS : Int := -1;   // Axis type: Invalid
      SPEED_AXIS : Int := 2;   // Axis type: Speed axis
      POSITIONING_AXIS : Int := 3;   // Axis type: Positioning axis
      SYNCHRONOUS_AXIS : Int := 4;   // Axis type: Synchronous axis
   END_VAR
BEGIN
   REGION HEADER
     //================================================================================
     // SIEMENS AG
     // (c)Copyright 2020 All Rights Reserved
     //--------------------------------------------------------------------------------
     // Library: LAnyAxis 
     // Tested with: S7-1515-2 PN
     // Engineering: TIA Portal V16
     // Restrictions: -
     // Requirements: S7-1500 FW 2.8.1
     // Functionality: Conversion DB_ANY --> TO_Axis
     // Support: tech.team.motioncontrol@siemens.com
     // Note: Parameter comments are only available in language 'English (United States)'
     //--------------------------------------------------------------------------------
     // Change log table:
     // Version  Date        Expert in charge  Changes applied
     // 01.00.00 10.03.2020  RS                First released version
     //================================================================================
   END_REGION

   REGION EXECUTE
     IF #Execute AND NOT #statExecuteOld THEN
       // Copy parameter
       #instMC.STW1 := #STW1;
       #instMC.STW1BitMask := #STW1BitMask;
       #instMC.STW2 := #STW2;
       #instMC.STW2BitMask := #STW2BitMask;

       // Check axis type
       CASE TypeOfDB(#Axis) OF
         TO_POSITIONINGAXIS:
           #statAxisType := #POSITIONING_AXIS;
           #statAxis := #Axis;

         TO_SYNCHRONOUSAXIS:
           #statAxisType := #SYNCHRONOUS_AXIS;
           #statAxis := #Axis;

         TO_SPEEDAXIS:
           #statAxisType := #SPEED_AXIS;
           #statAxis := #Axis;

         ELSE
           #statAxisType := #INVALID_AXIS;
           #statAxis := 0;
       END_CASE;

     ELSIF NOT #Execute AND (#statAxisType = #INVALID_AXIS) THEN
       #statAxisType := #IDLE;

       // Outputs
       #Done := FALSE;
       #Busy := FALSE;
       #CommandAborted := FALSE;
       #Error := FALSE;
       #ErrorID := 16#0000;
     END_IF;

     // Edge detection
     #statExecuteOld := #Execute;
   END_REGION

   CASE #statAxisType OF
     #IDLE:
       ;

     #POSITIONING_AXIS,
     #SYNCHRONOUS_AXIS,
     #SPEED_AXIS:
       REGION VALID_AXIS
         // Inputs
         #instMC.Execute := #Execute;

         // Call of MC instruction
         CASE #statAxisType OF
           #POSITIONING_AXIS:
             "LAnyAxis_UnpubSetAxisSTWPosAxis"(axis := #statAxis,
                                               instMC := #instMC);
           #SYNCHRONOUS_AXIS:
             "LAnyAxis_UnpubSetAxisSTWSyncAxis"(axis := #statAxis,
                                                instMC := #instMC);
           #SPEED_AXIS:
             #instMC(Axis := #statAxis);
         END_CASE;

         // Outputs
         #Done := #instMC.Done;
         #Busy := #instMC.Busy;
         #CommandAborted := #instMC.CommandAborted;
         #Error := #instMC.Error;
         #ErrorID := #instMC.ErrorId;

         // Status of MC instruction
         IF NOT #instMC.Done
           AND NOT #instMC.Busy
           AND NOT #instMC.CommandAborted
           AND NOT #instMC.Error
         THEN
           // Not active
           #statAxisType := #IDLE;
         END_IF;
       END_REGION

     ELSE
       REGION INVALID_AXIS
         // Outputs
         #Done := FALSE;
         #Busy := FALSE;
         #CommandAborted := FALSE;
         #Error := TRUE;
         #ErrorID := #ERROR_INVALID_TECHNOLOGY_OBJECT;
       END_REGION
   END_CASE;
END_FUNCTION_BLOCK

// folder: LAnyAxis_Blocks/InternalSubBlocks/MC_Halt

FUNCTION "LAnyAxis_UnpubHaltPosAxis" : Void   // FC30003, SCL
TITLE = LAnyAxis_UnpubHaltPosAxis
{ S7_Optimized_Access := 'TRUE' }
AUTHOR : tech.team.motioncontrol@siemens.com
FAMILY : AnyAxis
VERSION : 1.0
// Support: tech.team.motioncontrol@siemens.com
   VAR_INPUT
      axis : TO_PositioningAxis;   // Axis specification
   END_VAR
   VAR_IN_OUT
      instMC : MC_HALT;   // Instance of MC_Instruction
   END_VAR
   // Ret_Val : No return value
BEGIN
   // Call of MC_Instruction
   #instMC(Axis := #axis);
END_FUNCTION

FUNCTION "LAnyAxis_UnpubHaltSyncAxis" : Void   // FC30005, SCL
TITLE = LAnyAxis_UnpubHaltSyncAxis
{ S7_Optimized_Access := 'TRUE' }
AUTHOR : tech.team.motioncontrol@siemens.com
FAMILY : AnyAxis
VERSION : 1.0
// Support: tech.team.motioncontrol@siemens.com
   VAR_INPUT
      axis : TO_SynchronousAxis;   // Axis specification
   END_VAR
   VAR_IN_OUT
      instMC : MC_HALT;   // Instance of MC_Instruction
   END_VAR
   // Ret_Val : No return value
BEGIN
   // Call of MC_Instruction
   #instMC(Axis := #axis);
END_FUNCTION

// folder: LAnyAxis_Blocks/InternalSubBlocks/MC_Home

FUNCTION "LAnyAxis_UnpubHomeExtEncoder" : Void   // FC30058, SCL
TITLE = LAnyAxis_UnpubHomeExtEncoder
{ S7_Optimized_Access := 'TRUE' }
AUTHOR : tech.team.motioncontrol@siemens.com
FAMILY : AnyAxis
VERSION : 1.0
// Support: tech.team.motioncontrol@siemens.com
   VAR_INPUT
      axis : TO_ExternalEncoder;   // Axis specification
   END_VAR
   VAR_IN_OUT
      instMC : MC_HOME;   // Instance of MC_Instruction
   END_VAR
   // Ret_Val : No return value
BEGIN
   // Call of MC_Instruction
   #instMC(Axis := #axis);
END_FUNCTION

FUNCTION "LAnyAxis_UnpubHomePosAxis" : Void   // FC30059, SCL
TITLE = LAnyAxis_UnpubHomePosAxis
{ S7_Optimized_Access := 'TRUE' }
AUTHOR : tech.team.motioncontrol@siemens.com
FAMILY : AnyAxis
VERSION : 1.0
// Support: tech.team.motioncontrol@siemens.com
   VAR_INPUT
      axis : TO_PositioningAxis;   // Axis specification
   END_VAR
   VAR_IN_OUT
      instMC : MC_HOME;   // Instance of MC_Instruction
   END_VAR
   // Ret_Val : No return value
BEGIN
   // Call of MC_Instruction
   #instMC(Axis := #axis);
END_FUNCTION

FUNCTION "LAnyAxis_UnpubHomeSyncAxis" : Void   // FC30060, SCL
TITLE = LAnyAxis_UnpubHomeSyncAxis
{ S7_Optimized_Access := 'TRUE' }
AUTHOR : tech.team.motioncontrol@siemens.com
FAMILY : AnyAxis
VERSION : 1.0
// Support: tech.team.motioncontrol@siemens.com
   VAR_INPUT
      axis : TO_SynchronousAxis;   // Axis specification
   END_VAR
   VAR_IN_OUT
      instMC : MC_HOME;   // Instance of MC_Instruction
   END_VAR
   // Ret_Val : No return value
BEGIN
   // Call of MC_Instruction
   #instMC(Axis := #axis);
END_FUNCTION

// folder: LAnyAxis_Blocks/InternalSubBlocks/MC_MoveAbsolute

FUNCTION "LAnyAxis_UnpubMoveAbsoluteSyncAxis" : Void   // FC30007, SCL
TITLE = LAnyAxis_UnpubMoveAbsoluteSyncAxis
{ S7_Optimized_Access := 'TRUE' }
AUTHOR : tech.team.motioncontrol@siemens.com
FAMILY : AnyAxis
VERSION : 1.0
// Support: tech.team.motioncontrol@siemens.com
   VAR_INPUT
      axis : TO_SynchronousAxis;   // Axis specification
   END_VAR
   VAR_IN_OUT
      instMC : MC_MOVEABSOLUTE;   // Instance of MC_Instruction
   END_VAR
   // Ret_Val : No return value
BEGIN
   // Call of MC_Instruction
   #instMC(Axis := #axis);
END_FUNCTION

// folder: LAnyAxis_Blocks/InternalSubBlocks/MC_MoveJog

FUNCTION "LAnyAxis_UnpubMoveJogPosAxis" : Void   // FC30008, SCL
TITLE = LAnyAxis_UnpubMoveJogPosAxis
{ S7_Optimized_Access := 'TRUE' }
AUTHOR : tech.team.motioncontrol@siemens.com
FAMILY : AnyAxis
VERSION : 1.0
// Support: tech.team.motioncontrol@siemens.com
   VAR_INPUT
      axis : TO_PositioningAxis;   // Axis specification
   END_VAR
   VAR_IN_OUT
      instMC : MC_MOVEJOG;   // Instance of MC_Instruction
   END_VAR
   // Ret_Val : No return value
BEGIN
   // Call of MC_Instruction
   #instMC(Axis := #axis);
END_FUNCTION

FUNCTION "LAnyAxis_UnpubMoveJogSyncAxis" : Void   // FC30010, SCL
TITLE = LAnyAxis_UnpubMoveJogSyncAxis
{ S7_Optimized_Access := 'TRUE' }
AUTHOR : tech.team.motioncontrol@siemens.com
FAMILY : AnyAxis
VERSION : 1.0
// Support: tech.team.motioncontrol@siemens.com
   VAR_INPUT
      axis : TO_SynchronousAxis;   // Axis specification
   END_VAR
   VAR_IN_OUT
      instMC : MC_MOVEJOG;   // Instance of MC_Instruction
   END_VAR
   // Ret_Val : No return value
BEGIN
   // Call of MC_Instruction
   #instMC(Axis := #axis);
END_FUNCTION

// folder: LAnyAxis_Blocks/InternalSubBlocks/MC_MoveRelative

FUNCTION "LAnyAxis_UnpubMoveRelativeSyncAxis" : Void   // FC30012, SCL
TITLE = LAnyAxis_UnpubMoveRelativeSyncAxis
{ S7_Optimized_Access := 'TRUE' }
AUTHOR : tech.team.motioncontrol@siemens.com
FAMILY : AnyAxis
VERSION : 1.0
// Support: tech.team.motioncontrol@siemens.com
   VAR_INPUT
      axis : TO_SynchronousAxis;   // Axis specification
   END_VAR
   VAR_IN_OUT
      instMC : MC_MOVERELATIVE;   // Instance of MC_Instruction
   END_VAR
   // Ret_Val : No return value
BEGIN
   // Call of MC_Instruction
   #instMC(Axis := #axis);
END_FUNCTION

// folder: LAnyAxis_Blocks/InternalSubBlocks/MC_MoveSuperimposed

FUNCTION "LAnyAxis_UnpubMoveSuperimposedSyncAxis" : Void   // FC30014, SCL
TITLE = LAnyAxis_UnpubMoveSuperimposedSyncAxis
{ S7_Optimized_Access := 'TRUE' }
AUTHOR : tech.team.motioncontrol@siemens.com
FAMILY : AnyAxis
VERSION : 1.0
// Support: tech.team.motioncontrol@siemens.com
   VAR_INPUT
      axis : TO_SynchronousAxis;   // Axis specification
   END_VAR
   VAR_IN_OUT
      instMC : MC_MOVESUPERIMPOSED;   // Instance of MC_Instruction
   END_VAR
   // Ret_Val : No return value
BEGIN
   // Call of MC_Instruction
   #instMC(Axis := #axis);
END_FUNCTION

// folder: LAnyAxis_Blocks/InternalSubBlocks/MC_MoveVelocity

FUNCTION "LAnyAxis_UnpubMoveVelocityPosAxis" : Void   // FC30015, SCL
TITLE = LAnyAxis_UnpubMoveVelocityPosAxis
{ S7_Optimized_Access := 'TRUE' }
AUTHOR : tech.team.motioncontrol@siemens.com
FAMILY : AnyAxis
VERSION : 1.0
// Support: tech.team.motioncontrol@siemens.com
   VAR_INPUT
      axis : TO_PositioningAxis;   // Axis specification
   END_VAR
   VAR_IN_OUT
      instMC : MC_MOVEVELOCITY;   // Instance of MC_Instruction
   END_VAR
   // Ret_Val : No return value
BEGIN
   // Call of MC_Instruction
   #instMC(Axis := #axis);
END_FUNCTION

FUNCTION "LAnyAxis_UnpubMoveVelocitySyncAxis" : Void   // FC30017, SCL
TITLE = LAnyAxis_UnpubMoveVelocitySyncAxis
{ S7_Optimized_Access := 'TRUE' }
AUTHOR : tech.team.motioncontrol@siemens.com
FAMILY : AnyAxis
VERSION : 1.0
// Support: tech.team.motioncontrol@siemens.com
   VAR_INPUT
      axis : TO_SynchronousAxis;   // Axis specification
   END_VAR
   VAR_IN_OUT
      instMC : MC_MOVEVELOCITY;   // Instance of MC_Instruction
   END_VAR
   // Ret_Val : No return value
BEGIN
   // Call of MC_Instruction
   #instMC(Axis := #axis);
END_FUNCTION

// folder: LAnyAxis_Blocks/InternalSubBlocks/MC_Power

FUNCTION "LAnyAxis_UnpubPowerExtEncoder" : Void   // FC30018, SCL
TITLE = LAnyAxis_UnpubPowerExtEncoder
{ S7_Optimized_Access := 'TRUE' }
AUTHOR : tech.team.motioncontrol@siemens.com
FAMILY : AnyAxis
VERSION : 1.0
// Support: tech.team.motioncontrol@siemens.com
   VAR_INPUT
      axis : TO_ExternalEncoder;   // Axis specification
   END_VAR
   VAR_IN_OUT
      instMC : MC_POWER;   // Instance of MC_Instruction
   END_VAR
   // Ret_Val : No return value
BEGIN
   // Call of MC_Instruction
   #instMC(Axis := #axis);
END_FUNCTION

FUNCTION "LAnyAxis_UnpubPowerPosAxis" : Void   // FC30019, SCL
TITLE = LAnyAxis_UnpubPowerPosAxis
{ S7_Optimized_Access := 'TRUE' }
AUTHOR : tech.team.motioncontrol@siemens.com
FAMILY : AnyAxis
VERSION : 1.0
// Support: tech.team.motioncontrol@siemens.com
   VAR_INPUT
      axis : TO_PositioningAxis;   // Axis specification
   END_VAR
   VAR_IN_OUT
      instMC : MC_POWER;   // Instance of MC_Instruction
   END_VAR
   // Ret_Val : No return value
BEGIN
   // Call of MC_Instruction
   #instMC(Axis := #axis);
END_FUNCTION

FUNCTION "LAnyAxis_UnpubPowerSpeedAxis" : Void   // FC30020, SCL
TITLE = LAnyAxis_UnpubPowerSpeedAxis
{ S7_Optimized_Access := 'TRUE' }
AUTHOR : tech.team.motioncontrol@siemens.com
FAMILY : AnyAxis
VERSION : 1.0
// Support: tech.team.motioncontrol@siemens.com
   VAR_INPUT
      axis : TO_SpeedAxis;   // Axis specification
   END_VAR
   VAR_IN_OUT
      instMC : MC_POWER;   // Instance of MC_Instruction
   END_VAR
   // Ret_Val : No return value
BEGIN
   // Call of MC_Instruction
   #instMC(Axis := #axis);
END_FUNCTION

FUNCTION "LAnyAxis_UnpubPowerSyncAxis" : Void   // FC30021, SCL
TITLE = LAnyAxis_UnpubPowerSyncAxis
{ S7_Optimized_Access := 'TRUE' }
AUTHOR : tech.team.motioncontrol@siemens.com
FAMILY : AnyAxis
VERSION : 1.0
// Support: tech.team.motioncontrol@siemens.com
   VAR_INPUT
      axis : TO_SynchronousAxis;   // Axis specification
   END_VAR
   VAR_IN_OUT
      instMC : MC_POWER;   // Instance of MC_Instruction
   END_VAR
   // Ret_Val : No return value
BEGIN
   // Call of MC_Instruction
   #instMC(Axis := #axis);
END_FUNCTION

// folder: LAnyAxis_Blocks/InternalSubBlocks/MC_Reset

FUNCTION "LAnyAxis_UnpubResetExtEncoder" : Void   // FC30022, SCL
TITLE = LAnyAxis_UnpubResetExtEncoder
{ S7_Optimized_Access := 'TRUE' }
AUTHOR : tech.team.motioncontrol@siemens.com
FAMILY : AnyAxis
VERSION : 1.0
// Support: tech.team.motioncontrol@siemens.com
   VAR_INPUT
      axis : TO_ExternalEncoder;   // Axis specification
   END_VAR
   VAR_IN_OUT
      instMC : MC_RESET;   // Instance of MC_Instruction
   END_VAR
   // Ret_Val : No return value
BEGIN
   // Call of MC_Instruction
   #instMC(Axis := #axis);
END_FUNCTION

FUNCTION "LAnyAxis_UnpubResetSpeedAxis" : Void   // FC30024, SCL
TITLE = LAnyAxis_UnpubResetSpeedAxis
{ S7_Optimized_Access := 'TRUE' }
AUTHOR : tech.team.motioncontrol@siemens.com
FAMILY : AnyAxis
VERSION : 1.0
// Support: tech.team.motioncontrol@siemens.com
   VAR_INPUT
      axis : TO_SpeedAxis;   // Axis specification
   END_VAR
   VAR_IN_OUT
      instMC : MC_RESET;   // Instance of MC_Instruction
   END_VAR
   // Ret_Val : No return value
BEGIN
   // Call of MC_Instruction
   #instMC(Axis := #axis);
END_FUNCTION

FUNCTION "LAnyAxis_UnpubResetSyncAxis" : Void   // FC30025, SCL
TITLE = LAnyAxis_UnpubResetSyncAxis
{ S7_Optimized_Access := 'TRUE' }
AUTHOR : tech.team.motioncontrol@siemens.com
FAMILY : AnyAxis
VERSION : 1.0
// Support: tech.team.motioncontrol@siemens.com
   VAR_INPUT
      axis : TO_SynchronousAxis;   // Axis specification
   END_VAR
   VAR_IN_OUT
      instMC : MC_RESET;   // Instance of MC_Instruction
   END_VAR
   // Ret_Val : No return value
BEGIN
   // Call of MC_Instruction
   #instMC(Axis := #axis);
END_FUNCTION

FUNCTION "LAnyAxis_UnpubResetPosAxis" : Void   // FC30071, SCL
TITLE = LAnyAxis_UnpubResetPosAxis
{ S7_Optimized_Access := 'TRUE' }
AUTHOR : tech.team.motioncontrol@siemens.com
FAMILY : AnyAxis
VERSION : 1.0
// Support: tech.team.motioncontrol@siemens.com
   VAR_INPUT
      axis : TO_PositioningAxis;   // Axis specification
   END_VAR
   VAR_IN_OUT
      instMC : MC_RESET;   // Instance of MC_Instruction
   END_VAR
   // Ret_Val : No return value
BEGIN
   // Call of MC_Instruction
   #instMC(Axis := #axis);
END_FUNCTION

// folder: LAnyAxis_Blocks/InternalSubBlocks/MC_SetAxisSTW

FUNCTION "LAnyAxis_UnpubSetAxisSTWPosAxis" : Void   // FC30026, SCL
TITLE = LAnyAxis_UnpubSetAxisSTWPosAxis
{ S7_Optimized_Access := 'TRUE' }
AUTHOR : tech.team.motioncontrol@siemens.com
FAMILY : AnyAxis
VERSION : 1.0
// Support: tech.team.motioncontrol@siemens.com
   VAR_INPUT
      axis : TO_PositioningAxis;   // Axis specification
   END_VAR
   VAR_IN_OUT
      instMC : MC_SETAXISSTW;   // Instance of MC_Instruction
   END_VAR
   // Ret_Val : No return value
BEGIN
   // Call of MC_Instruction
   #instMC(Axis := #axis);
END_FUNCTION

FUNCTION "LAnyAxis_UnpubSetAxisSTWSyncAxis" : Void   // FC30028, SCL
TITLE = LAnyAxis_UnpubSetAxisSTWSyncAxis
{ S7_Optimized_Access := 'TRUE' }
AUTHOR : tech.team.motioncontrol@siemens.com
FAMILY : AnyAxis
VERSION : 1.0
// Support: tech.team.motioncontrol@siemens.com
   VAR_INPUT
      axis : TO_SynchronousAxis;   // Axis specification
   END_VAR
   VAR_IN_OUT
      instMC : MC_SETAXISSTW;   // Instance of MC_Instruction
   END_VAR
   // Ret_Val : No return value
BEGIN
   // Call of MC_Instruction
   #instMC(Axis := #axis);
END_FUNCTION

// folder: LAnyAxis_Blocks/LAnyAxis_MC_SynchronousMotion

FUNCTION_BLOCK "LAnyAxis_MC_GearIn"   // FB30020, SCL
TITLE = LAnyAxis_MC_GearIn
{ S7_Optimized_Access := 'TRUE' }
AUTHOR : tech.team.motioncontrol@siemens.com
FAMILY : AnyAxis
VERSION : 1.0
// Support: tech.team.motioncontrol@siemens.com 
// See corresponding MC_ instruction in TIA Portal help (information system)
   VAR_INPUT
      Master : DB_ANY;   // See corresponding parameter of MC_ instruction in TIA Portal help (information system)
      Slave : DB_ANY;   // See corresponding parameter of MC_ instruction in TIA Portal help (information system)
      Execute : Bool;   // See corresponding parameter of MC_ instruction in TIA Portal help (information system)
      RatioNumerator : DInt := 1;   // See corresponding parameter of MC_ instruction in TIA Portal help (information system)
      RatioDenominator : DInt := 1;   // See corresponding parameter of MC_ instruction in TIA Portal help (information system)
      Acceleration : LReal := -1.0;   // See corresponding parameter of MC_ instruction in TIA Portal help (information system)
      Deceleration : LReal := -1.0;   // See corresponding parameter of MC_ instruction in TIA Portal help (information system)
      Jerk : LReal := -1.0;   // See corresponding parameter of MC_ instruction in TIA Portal help (information system)
   END_VAR
   VAR_OUTPUT
      InGear : Bool;   // See corresponding parameter of MC_ instruction in TIA Portal help (information system)
      Busy : Bool;   // See corresponding parameter of MC_ instruction in TIA Portal help (information system)
      CommandAborted : Bool;   // See corresponding parameter of MC_ instruction in TIA Portal help (information system)
      Error : Bool;   // See corresponding parameter of MC_ instruction in TIA Portal help (information system)
      ErrorID : Word;   // See corresponding parameter of MC_ instruction in TIA Portal help (information system)
   END_VAR
   VAR
      instMC : MC_GEARIN;   // Instance of MC_Instruction
      statExecuteOld : Bool;   // Old value of execute
      statAxis : DB_ANY;   // Internal variable of axis
      statAxisType : Int;   // Actual state / axis type
      statMaster : DB_ANY;   // Internal variable of Master
      statMasterType : Int;   // Type of master axis
   END_VAR
   VAR CONSTANT
      ERROR_INVALID_TECHNOLOGY_OBJECT : Word := 16#8002;   // See corresponding parameter of MC_ instruction in TIA Portal help (information system)
      IDLE : Int := 0;   // State idle
      INVALID_AXIS : Int := -1;   // Axis type: Invalid
      INVALID_MASTER : Int := -2;   // Invalid master type
      EXTERNAL_ENCODER : Int := 1;   // Axis type: External encoder
      POSITIONING_AXIS : Int := 3;   // Axis type: Positioning axis
      SYNCHRONOUS_AXIS : Int := 4;   // Axis type: Synchronous axis
   END_VAR
BEGIN
   REGION HEADER
     //================================================================================
     // SIEMENS AG
     // (c)Copyright 2020 All Rights Reserved
     //--------------------------------------------------------------------------------
     // Library: LAnyAxis 
     // Tested with: S7-1515-2 PN
     // Engineering: TIA Portal V16
     // Restrictions: -
     // Requirements: S7-1500 FW 2.8.1
     // Functionality: Conversion DB_ANY --> TO_Axis
     // Support: tech.team.motioncontrol@siemens.com
     // Note: Parameter comments are only available in language 'English (United States)'
     //--------------------------------------------------------------------------------
     // Change log table:
     // Version  Date        Expert in charge  Changes applied
     // 01.00.00 10.03.2020  RS                First released version
     //================================================================================
   END_REGION

   REGION EXECUTE
     IF #Execute AND NOT #statExecuteOld THEN
       // Copy parameter
       #instMC.RatioNumerator := #RatioNumerator;
       #instMC.RatioDenominator := #RatioDenominator;
       #instMC.Acceleration := #Acceleration;
       #instMC.Deceleration := #Deceleration;
       #instMC.Jerk := #Jerk;

       // Check axis type
       CASE TypeOfDB(#Slave) OF
         TO_SYNCHRONOUSAXIS:
           #statAxisType := #SYNCHRONOUS_AXIS;
           #statAxis := #Slave;

           // Check master type
           CASE TypeOfDB(#Master) OF
             TO_POSITIONINGAXIS:
               #statMasterType := #POSITIONING_AXIS;
               #statMaster := #Master;

             TO_SYNCHRONOUSAXIS:
               #statMasterType := #SYNCHRONOUS_AXIS;
               #statMaster := #Master;

             TO_EXTERNALENCODER:
               #statMasterType := #EXTERNAL_ENCODER;
               #statMaster := #Master;

             ELSE
               // Invalid master
               #statMasterType := #INVALID_AXIS;
               #statMaster := 0;

               #statAxisType := #INVALID_MASTER;
           END_CASE;

         ELSE
           #statAxisType := #INVALID_AXIS;
           #statAxis := 0;
       END_CASE;

     ELSIF NOT #Execute AND (#statAxisType < #IDLE) THEN
       #statAxisType := #IDLE;

       // Outputs
       #InGear := FALSE;
       #Busy := FALSE;
       #CommandAborted := FALSE;
       #Error := FALSE;
       #ErrorID := 16#0000;
     END_IF;

     // Edge detection
     #statExecuteOld := #Execute;
   END_REGION

   CASE #statAxisType OF
     #IDLE:
       ;

     #SYNCHRONOUS_AXIS:
       REGION VALID_AXIS
         // Inputs
         #instMC.Execute := #Execute;

         // Call of MC instruction
         CASE #statMasterType OF
           #POSITIONING_AXIS:
             "LAnyAxis_UnpubGearInMasterPosAxis"(slave := #statAxis,
                                                 master := #statMaster,
                                                 instMC := #instMC);
           #SYNCHRONOUS_AXIS:
             "LAnyAxis_UnpubGearInMasterSyncAxis"(slave := #statAxis,
                                                  master := #statMaster,
                                                  instMC := #instMC);
           #EXTERNAL_ENCODER:
             "LAnyAxis_UnpubGearInMasterExtEncoder"(slave := #statAxis,
                                                    master := #statMaster,
                                                    instMC := #instMC);
         END_CASE;

         // Outputs
         #InGear := #instMC.InGear;
         #Busy := #instMC.Busy;
         #CommandAborted := #instMC.CommandAborted;
         #Error := #instMC.Error;
         #ErrorID := #instMC.ErrorId;

         // Status of MC instruction
         IF NOT #instMC.Busy
           AND NOT #instMC.CommandAborted
           AND NOT #instMC.Error
         THEN
           // Not active
           #statAxisType := #IDLE;
         END_IF;
       END_REGION

     ELSE
       REGION INVALID_TECHNOLOGY_OBJECT
         // Outputs
         #InGear := FALSE;
         #Busy := FALSE;
         #CommandAborted := FALSE;
         #Error := TRUE;
         #ErrorID := #ERROR_INVALID_TECHNOLOGY_OBJECT;
       END_REGION
   END_CASE;
END_FUNCTION_BLOCK

// folder: LAnyAxis_Blocks/LAnyAxis_MC_SynchronousMotion/InternalDummyBlocks

FUNCTION_BLOCK "LAnyAxis_MC_GearInPos"   // FB30021, SCL
TITLE = LAnyAxis_MC_GearInPos
{ S7_Optimized_Access := 'TRUE' }
AUTHOR : tech.team.motioncontrol@siemens.com
FAMILY : AnyAxis
VERSION : 1.0
// Support: tech.team.motioncontrol@siemens.com 
// This block is for internal use only
   VAR_INPUT
      Master : DB_ANY;   // See corresponding parameter of MC_ instruction in TIA Portal help (information system)
      Slave : DB_ANY;   // See corresponding parameter of MC_ instruction in TIA Portal help (information system)
      Execute : Bool;   // See corresponding parameter of MC_ instruction in TIA Portal help (information system)
      RatioNumerator : DInt := 1;   // See corresponding parameter of MC_ instruction in TIA Portal help (information system)
      RatioDenominator : DInt := 1;   // See corresponding parameter of MC_ instruction in TIA Portal help (information system)
      MasterSyncPosition : LReal;   // See corresponding parameter of MC_ instruction in TIA Portal help (information system)
      SlaveSyncPosition : LReal;   // See corresponding parameter of MC_ instruction in TIA Portal help (information system)
      SyncProfileReference : DInt := 1;   // See corresponding parameter of MC_ instruction in TIA Portal help (information system)
      MasterStartDistance : LReal := 1.0;   // See corresponding parameter of MC_ instruction in TIA Portal help (information system)
      Velocity : LReal := -1.0;   // See corresponding parameter of MC_ instruction in TIA Portal help (information system)
      Acceleration : LReal := -1.0;   // See corresponding parameter of MC_ instruction in TIA Portal help (information system)
      Deceleration : LReal := -1.0;   // See corresponding parameter of MC_ instruction in TIA Portal help (information system)
      Jerk : LReal := -1.0;   // See corresponding parameter of MC_ instruction in TIA Portal help (information system)
      SyncDirection : DInt := 3;   // See corresponding parameter of MC_ instruction in TIA Portal help (information system)
   END_VAR
   VAR_OUTPUT
      StartSync : Bool;   // See corresponding parameter of MC_ instruction in TIA Portal help (information system)
      InSync : Bool;   // See corresponding parameter of MC_ instruction in TIA Portal help (information system)
      Busy : Bool;   // See corresponding parameter of MC_ instruction in TIA Portal help (information system)
      CommandAborted : Bool;   // See corresponding parameter of MC_ instruction in TIA Portal help (information system)
      Error : Bool;   // See corresponding parameter of MC_ instruction in TIA Portal help (information system)
      ErrorID : Word;   // See corresponding parameter of MC_ instruction in TIA Portal help (information system)
   END_VAR
   VAR CONSTANT
      ERROR_INVALID_TECHNOLOGY_OBJECT : Word := 16#8002;   // See corresponding parameter of MC_ instruction in TIA Portal help (information system)
   END_VAR
BEGIN
   REGION HEADER
     //================================================================================
     // SIEMENS AG
     // (c)Copyright 2020 All Rights Reserved
     //--------------------------------------------------------------------------------
     // Library: LAnyAxis 
     // Tested with: S7-1515-2 PN
     // Engineering: TIA Portal V16
     // Restrictions: -
     // Requirements: S7-1500 FW 2.8.1
     // Functionality: Conversion DB_ANY --> TO_Axis
     // Support: tech.team.motioncontrol@siemens.com
     // Note: Parameter comments are only available in language 'English (United States)'
     //--------------------------------------------------------------------------------
     // Change log table:
     // Version  Date        Expert in charge  Changes applied
     // 01.00.00 10.03.2020  RS                First released version
     //================================================================================
   END_REGION

   #StartSync := FALSE;
   #InSync := FALSE;
   #Busy := FALSE;
   #CommandAborted := FALSE;

   IF #Execute THEN
     #Error := TRUE;
     #ErrorID := #ERROR_INVALID_TECHNOLOGY_OBJECT;
   ELSE
     #Error := FALSE;
     #ErrorID := 16#0000;
   END_IF;
END_FUNCTION_BLOCK

FUNCTION_BLOCK "LAnyAxis_MC_PhasingRelative"   // FB30022, SCL
TITLE = LAnyAxis_MC_PhasingRelative
{ S7_Optimized_Access := 'TRUE' }
AUTHOR : tech.team.motioncontrol@siemens.com
FAMILY : AnyAxis
VERSION : 1.1
// Support: tech.team.motioncontrol@siemens.com 
// This block is for internal use only
   VAR_INPUT
      Master : DB_ANY;   // See corresponding parameter of MC_ instruction in TIA Portal help (information system)
      Slave : DB_ANY;   // See corresponding parameter of MC_ instruction in TIA Portal help (information system)
      Execute : Bool;   // See corresponding parameter of MC_ instruction in TIA Portal help (information system)
      PhaseShift : LReal;   // See corresponding parameter of MC_ instruction in TIA Portal help (information system)
      Velocity : LReal := -1.0;   // See corresponding parameter of MC_ instruction in TIA Portal help (information system)
      Acceleration : LReal := -1.0;   // See corresponding parameter of MC_ instruction in TIA Portal help (information system)
      Deceleration : LReal := -1.0;   // See corresponding parameter of MC_ instruction in TIA Portal help (information system)
      Jerk : LReal := -1.0;   // See corresponding parameter of MC_ instruction in TIA Portal help (information system)
      ProfileReference : DInt;   // See corresponding parameter of MC_ instruction in TIA Portal help (information system)
      PhasingDistance : LReal;   // See corresponding parameter of MC_ instruction in TIA Portal help (information system)
      StartPosition : LReal;   // See corresponding parameter of MC_ instruction in TIA Portal help (information system)
      Direction : DInt := 3;   // See corresponding parameter of MC_ instruction in TIA Portal help (information system)
   END_VAR
   VAR_OUTPUT
      Done : Bool;   // See corresponding parameter of MC_ instruction in TIA Portal help (information system)
      Busy : Bool;   // See corresponding parameter of MC_ instruction in TIA Portal help (information system)
      CommandAborted : Bool;   // See corresponding parameter of MC_ instruction in TIA Portal help (information system)
      Error : Bool;   // See corresponding parameter of MC_ instruction in TIA Portal help (information system)
      ErrorID : Word;   // See corresponding parameter of MC_ instruction in TIA Portal help (information system)
      CoveredPhaseShift : LReal;   // See corresponding parameter of MC_ instruction in TIA Portal help (information system)
      StartPhasing : Bool;   // See corresponding parameter of MC_ instruction in TIA Portal help (information system)
   END_VAR
   VAR CONSTANT
      ERROR_INVALID_TECHNOLOGY_OBJECT : Word := 16#8002;   // See corresponding parameter of MC_ instruction in TIA Portal help (information system)
   END_VAR
BEGIN
   REGION HEADER
     //================================================================================
     // SIEMENS AG
     // (c)Copyright 2021 All Rights Reserved
     //--------------------------------------------------------------------------------
     // Library: LAnyAxis 
     // Tested with: S7-1515-2 PN
     // Engineering: TIA Portal V17
     // Restrictions: -
     // Requirements: S7-1500 FW 2.9 
     // Functionality: Conversion DB_ANY --> TO_Axis
     // Support: tech.team.motioncontrol@siemens.com
     // Note: Parameter comments are only available in language 'English (United States)'
     //--------------------------------------------------------------------------------
     // Change log table:
     // Version  Date        Expert in charge  Changes applied
     // 01.00.00 10.03.2020  RS                First released version
     // 01.01.00 24.02.2021  RS                Update MC V6.0
     //================================================================================
   END_REGION

   #Done := FALSE;
   #Busy := FALSE;
   #CommandAborted := FALSE;
   #CoveredPhaseShift := 0.0;
   #StartPhasing := FALSE;

   IF #Execute THEN
     #Error := TRUE;
     #ErrorID := #ERROR_INVALID_TECHNOLOGY_OBJECT;
   ELSE
     #Error := FALSE;
     #ErrorID := 16#0000;
   END_IF;
END_FUNCTION_BLOCK

FUNCTION_BLOCK "LAnyAxis_MC_PhasingAbsolute"   // FB30023, SCL
TITLE = LAnyAxis_MC_PhasingAbsolute
{ S7_Optimized_Access := 'TRUE' }
AUTHOR : tech.team.motioncontrol@siemens.com
FAMILY : AnyAxis
VERSION : 1.1
// Support: tech.team.motioncontrol@siemens.com 
// This block is for internal use only
   VAR_INPUT
      Master : DB_ANY;   // See corresponding parameter of MC_ instruction in TIA Portal help (information system)
      Slave : DB_ANY;   // See corresponding parameter of MC_ instruction in TIA Portal help (information system)
      Execute : Bool;   // See corresponding parameter of MC_ instruction in TIA Portal help (information system)
      PhaseShift : LReal;   // See corresponding parameter of MC_ instruction in TIA Portal help (information system)
      Velocity : LReal := -1.0;   // See corresponding parameter of MC_ instruction in TIA Portal help (information system)
      Acceleration : LReal := -1.0;   // See corresponding parameter of MC_ instruction in TIA Portal help (information system)
      Deceleration : LReal := -1.0;   // See corresponding parameter of MC_ instruction in TIA Portal help (information system)
      Jerk : LReal := -1.0;   // See corresponding parameter of MC_ instruction in TIA Portal help (information system)
      ProfileReference : DInt;   // See corresponding parameter of MC_ instruction in TIA Portal help (information system)
      PhasingDistance : LReal;   // See corresponding parameter of MC_ instruction in TIA Portal help (information system)
      StartPosition : LReal;   // See corresponding parameter of MC_ instruction in TIA Portal help (information system)
      Direction : DInt := 3;   // See corresponding parameter of MC_ instruction in TIA Portal help (information system)
   END_VAR
   VAR_OUTPUT
      Done : Bool;   // See corresponding parameter of MC_ instruction in TIA Portal help (information system)
      Busy : Bool;   // See corresponding parameter of MC_ instruction in TIA Portal help (information system)
      CommandAborted : Bool;   // See corresponding parameter of MC_ instruction in TIA Portal help (information system)
      Error : Bool;   // See corresponding parameter of MC_ instruction in TIA Portal help (information system)
      ErrorID : Word;   // See corresponding parameter of MC_ instruction in TIA Portal help (information system)
      AbsolutePhaseShift : LReal;   // See corresponding parameter of MC_ instruction in TIA Portal help (information system)
      StartPhasing : Bool;   // See corresponding parameter of MC_ instruction in TIA Portal help (information system)
   END_VAR
   VAR CONSTANT
      ERROR_INVALID_TECHNOLOGY_OBJECT : Word := 16#8002;   // See corresponding parameter of MC_ instruction in TIA Portal help (information system)
   END_VAR
BEGIN
   REGION HEADER
     //================================================================================
     // SIEMENS AG
     // (c)Copyright 2021 All Rights Reserved
     //--------------------------------------------------------------------------------
     // Library: LAnyAxis 
     // Tested with: S7-1515-2 PN
     // Engineering: TIA Portal V17
     // Restrictions: -
     // Requirements: S7-1500 FW 2.9 
     // Functionality: Conversion DB_ANY --> TO_Axis
     // Support: tech.team.motioncontrol@siemens.com
     // Note: Parameter comments are only available in language 'English (United States)'
     //--------------------------------------------------------------------------------
     // Change log table:
     // Version  Date        Expert in charge  Changes applied
     // 01.00.00 10.03.2020  RS                First released version
     // 01.01.00 24.02.2021  RS                Update MC V6.0
     //================================================================================
   END_REGION

   #Done := FALSE;
   #Busy := FALSE;
   #CommandAborted := FALSE;
   #AbsolutePhaseShift := 0.0;
   #StartPhasing := FALSE;

   IF #Execute THEN
     #Error := TRUE;
     #ErrorID := #ERROR_INVALID_TECHNOLOGY_OBJECT;
   ELSE
     #Error := FALSE;
     #ErrorID := 16#0000;
   END_IF;
END_FUNCTION_BLOCK

FUNCTION_BLOCK "LAnyAxis_MC_CamIn"   // FB30024, SCL
TITLE = LAnyAxis_MC_CamIn
{ S7_Optimized_Access := 'TRUE' }
AUTHOR : tech.team.motioncontrol@siemens.com
FAMILY : AnyAxis
VERSION : 1.1
// Support: tech.team.motioncontrol@siemens.com 
// This block is for internal use only
   VAR_INPUT
      Master : DB_ANY;   // See corresponding parameter of MC_ instruction in TIA Portal help (information system)
      Slave : DB_ANY;   // See corresponding parameter of MC_ instruction in TIA Portal help (information system)
      Cam : DB_ANY;   // See corresponding parameter of MC_ instruction in TIA Portal help (information system)
      Execute : Bool;   // See corresponding parameter of MC_ instruction in TIA Portal help (information system)
      MasterOffset : LReal;   // See corresponding parameter of MC_ instruction in TIA Portal help (information system)
      SlaveOffset : LReal;   // See corresponding parameter of MC_ instruction in TIA Portal help (information system)
      MasterScaling : LReal := 1.0;   // See corresponding parameter of MC_ instruction in TIA Portal help (information system)
      SlaveScaling : LReal := 1.0;   // See corresponding parameter of MC_ instruction in TIA Portal help (information system)
      MasterSyncPosition : LReal;   // See corresponding parameter of MC_ instruction in TIA Portal help (information system)
      SyncProfileReference : DInt := 1;   // See corresponding parameter of MC_ instruction in TIA Portal help (information system)
      MasterStartDistance : LReal;   // See corresponding parameter of MC_ instruction in TIA Portal help (information system)
      Velocity : LReal := -1.0;   // See corresponding parameter of MC_ instruction in TIA Portal help (information system)
      Acceleration : LReal := -1.0;   // See corresponding parameter of MC_ instruction in TIA Portal help (information system)
      Deceleration : LReal := -1.0;   // See corresponding parameter of MC_ instruction in TIA Portal help (information system)
      Jerk : LReal := -1.0;   // See corresponding parameter of MC_ instruction in TIA Portal help (information system)
      ApplicationMode : DInt;   // See corresponding parameter of MC_ instruction in TIA Portal help (information system)
      SyncDirection : DInt := 3;   // See corresponding parameter of MC_ instruction in TIA Portal help (information system)
   END_VAR
   VAR_OUTPUT
      StartSync : Bool;   // See corresponding parameter of MC_ instruction in TIA Portal help (information system)
      InSync : Bool;   // See corresponding parameter of MC_ instruction in TIA Portal help (information system)
      Busy : Bool;   // See corresponding parameter of MC_ instruction in TIA Portal help (information system)
      CommandAborted : Bool;   // See corresponding parameter of MC_ instruction in TIA Portal help (information system)
      Error : Bool;   // See corresponding parameter of MC_ instruction in TIA Portal help (information system)
      ErrorID : Word;   // See corresponding parameter of MC_ instruction in TIA Portal help (information system)
      EndOfProfile : Bool;   // See corresponding parameter of MC_ instruction in TIA Portal help (information system)
   END_VAR
   VAR CONSTANT
      ERROR_INVALID_TECHNOLOGY_OBJECT : Word := 16#8002;   // Illegal specification of the technology object. Check the specification of the technology object for the "Axis", "Master" or "Cam" parameter.
   END_VAR
BEGIN
   REGION HEADER
     //================================================================================
     // SIEMENS AG
     // (c)Copyright 2021 All Rights Reserved
     //--------------------------------------------------------------------------------
     // Library: LAnyAxis 
     // Tested with: S7-1515-2 PN
     // Engineering: TIA Portal V17
     // Restrictions: -
     // Requirements: S7-1500 FW 2.9 
     // Functionality: Conversion DB_ANY --> TO_Axis
     // Support: tech.team.motioncontrol@siemens.com
     // Note: Parameter comments are only available in language 'English (United States)'
     //--------------------------------------------------------------------------------
     // Change log table:
     // Version  Date        Expert in charge  Changes applied
     // 01.00.00 10.03.2020  RS                First released version
     // 01.01.00 24.02.2021  RS                Update MC V6.0
     //================================================================================
   END_REGION

   #StartSync := FALSE;
   #InSync := FALSE;
   #Busy := FALSE;
   #CommandAborted := FALSE;
   #EndOfProfile := FALSE;

   IF #Execute THEN
     #Error := TRUE;
     #ErrorID := #ERROR_INVALID_TECHNOLOGY_OBJECT;
   ELSE
     #Error := FALSE;
     #ErrorID := 16#0000;
   END_IF;
END_FUNCTION_BLOCK

FUNCTION_BLOCK "LAnyAxis_MC_SynchronizedMotionSimulation"   // FB30025, SCL
TITLE = LAnyAxis_MC_SynchronizedMotionSimulation
{ S7_Optimized_Access := 'TRUE' }
AUTHOR : tech.team.motioncontrol@siemens.com
FAMILY : AnyAxis
VERSION : 1.0
// Support: tech.team.motioncontrol@siemens.com 
// This block is for internal use only
   VAR_INPUT
      Slave : DB_ANY;   // See corresponding parameter of MC_ instruction in TIA Portal help (information system)
      Enable : Bool;   // See corresponding parameter of MC_ instruction in TIA Portal help (information system)
   END_VAR
   VAR_OUTPUT
      InSimulation : Bool;   // See corresponding parameter of MC_ instruction in TIA Portal help (information system)
      Busy : Bool;   // See corresponding parameter of MC_ instruction in TIA Portal help (information system)
      Error : Bool;   // See corresponding parameter of MC_ instruction in TIA Portal help (information system)
      ErrorID : Word;   // See corresponding parameter of MC_ instruction in TIA Portal help (information system)
   END_VAR
   VAR CONSTANT
      ERROR_INVALID_TECHNOLOGY_OBJECT : Word := 16#8002;   // See corresponding parameter of MC_ instruction in TIA Portal help (information system)
   END_VAR
BEGIN
   REGION HEADER
     //================================================================================
     // SIEMENS AG
     // (c)Copyright 2020 All Rights Reserved
     //--------------------------------------------------------------------------------
     // Library: LAnyAxis 
     // Tested with: S7-1515-2 PN
     // Engineering: TIA Portal V16
     // Restrictions: -
     // Requirements: S7-1500 FW 2.8.1
     // Functionality: Conversion DB_ANY --> TO_Axis
     // Support: tech.team.motioncontrol@siemens.com
     // Note: Parameter comments are only available in language 'English (United States)'
     //--------------------------------------------------------------------------------
     // Change log table:
     // Version  Date        Expert in charge  Changes applied
     // 01.00.00 10.03.2020  RS                First released version
     //================================================================================
   END_REGION

   #Busy := FALSE;
   #InSimulation := FALSE;

   IF #Enable THEN
     #Error := TRUE;
     #ErrorID := #ERROR_INVALID_TECHNOLOGY_OBJECT;
   ELSE
     #Error := TRUE;
     #ErrorID := 16#0000;
   END_IF;
END_FUNCTION_BLOCK

